(* Logix 5000 project; controller reports 1756-L63 rev 20.11; software revision 20.04; part 21 of 52 *)

        [1300].log_data[12].valid := 1, [1300].log_data[13].valid := 1, [1300].log_data[14].valid := 1, [1300].log_data[15].valid := 1, [1300].log_data[16].valid := 1, [1300].log_data[17].valid := 1, [1300].log_data[18].valid := 1, [1300].log_data[19].valid := 1, [1300].time.Year := 2023, [1300].time.Month := 1, [1300].time.Day := 14, [1300].time.Hour := 4, [1300].time.Minute := 44, [1300].time.Second := 59, [1301].log_data[0].min := 1.0, [1301].log_data[0].max := 1.0, [1301].log_data[0].total := 300.0, [1301].log_data[0].time := 300.0, [1301].log_data[0].minminute := 45, [1301].log_data[0].maxminute := 45, [1301].log_data[0].valid := 1, [1301].log_data[1].valid := 1, [1301].log_data[2].valid := 1, [1301].log_data[3].valid := 1, [1301].log_data[4].valid := 1, [1301].log_data[5].valid := 1, [1301].log_data[6].valid := 1, [1301].log_data[7].valid := 1, [1301].log_data[8].valid := 1, [1301].log_data[9].valid := 1, [1301].log_data[10].valid := 1, [1301].log_data[11].valid := 1, [1301].log_data[12].valid := 1, [1301].log_data[13].valid := 1, [1301].log_data[14].valid := 1, [1301].log_data[15].valid := 1, [1301].log_data[16].valid := 1, [1301].log_data[17].valid := 1, [1301].log_data[18].valid := 1, [1301].log_data[19].valid := 1, [1301].time.Year := 2023, [1301].time.Month := 1, [1301].time.Day := 14, [1301].time.Hour := 4, [1301].time.Minute := 49, [1301].time.Second := 59, [1302].log_data[0].min := 1.0, [1302].log_data[0].max := 1.0, [1302].log_data[0].total := 300.0, [1302].log_data[0].time := 300.0, [1302].log_data[0].minminute := 50, [1302].log_data[0].maxminute := 50, [1302].log_data[0].valid := 1, [1302].log_data[1].valid := 1, [1302].log_data[2].valid := 1, [1302].log_data[3].valid := 1, [1302].log_data[4].valid := 1, [1302].log_data[5].valid := 1, [1302].log_data[6].valid := 1, [1302].log_data[7].valid := 1,
        [1302].log_data[8].valid := 1, [1302].log_data[9].valid := 1, [1302].log_data[10].valid := 1, [1302].log_data[11].valid := 1, [1302].log_data[12].valid := 1, [1302].log_data[13].valid := 1, [1302].log_data[14].valid := 1, [1302].log_data[15].valid := 1, [1302].log_data[16].valid := 1, [1302].log_data[17].valid := 1, [1302].log_data[18].valid := 1, [1302].log_data[19].valid := 1, [1302].time.Year := 2023, [1302].time.Month := 1, [1302].time.Day := 14, [1302].time.Hour := 4, [1302].time.Minute := 54, [1302].time.Second := 59, [1303].log_data[0].min := 1.0, [1303].log_data[0].max := 1.0, [1303].log_data[0].total := 300.0, [1303].log_data[0].time := 300.0, [1303].log_data[0].minminute := 55, [1303].log_data[0].maxminute := 55, [1303].log_data[0].valid := 1, [1303].log_data[1].valid := 1, [1303].log_data[2].valid := 1, [1303].log_data[3].valid := 1, [1303].log_data[4].valid := 1, [1303].log_data[5].valid := 1, [1303].log_data[6].valid := 1, [1303].log_data[7].valid := 1, [1303].log_data[8].valid := 1, [1303].log_data[9].valid := 1, [1303].log_data[10].valid := 1, [1303].log_data[11].valid := 1, [1303].log_data[12].valid := 1, [1303].log_data[13].valid := 1, [1303].log_data[14].valid := 1, [1303].log_data[15].valid := 1, [1303].log_data[16].valid := 1, [1303].log_data[17].valid := 1, [1303].log_data[18].valid := 1, [1303].log_data[19].valid := 1, [1303].time.Year := 2023, [1303].time.Month := 1, [1303].time.Day := 14, [1303].time.Hour := 4, [1303].time.Minute := 59, [1303].time.Second := 59, [1304].log_data[0].min := 1.0, [1304].log_data[0].max := 1.0, [1304].log_data[0].total := 300.0, [1304].log_data[0].time := 300.0, [1304].log_data[0].valid := 1, [1304].log_data[1].valid := 1, [1304].log_data[2].valid := 1, [1304].log_data[3].valid := 1, [1304].log_data[4].valid := 1, [1304].log_data[5].valid := 1,
        [1304].log_data[6].valid := 1, [1304].log_data[7].valid := 1, [1304].log_data[8].valid := 1, [1304].log_data[9].valid := 1, [1304].log_data[10].valid := 1, [1304].log_data[11].valid := 1, [1304].log_data[12].valid := 1, [1304].log_data[13].valid := 1, [1304].log_data[14].valid := 1, [1304].log_data[15].valid := 1, [1304].log_data[16].valid := 1, [1304].log_data[17].valid := 1, [1304].log_data[18].valid := 1, [1304].log_data[19].valid := 1, [1304].time.Year := 2023, [1304].time.Month := 1, [1304].time.Day := 14, [1304].time.Hour := 5, [1304].time.Minute := 4, [1304].time.Second := 59, [1305].log_data[0].min := 1.0, [1305].log_data[0].max := 1.0, [1305].log_data[0].total := 300.0, [1305].log_data[0].time := 300.0, [1305].log_data[0].minminute := 5, [1305].log_data[0].maxminute := 5, [1305].log_data[0].valid := 1, [1305].log_data[1].valid := 1, [1305].log_data[2].valid := 1, [1305].log_data[3].valid := 1, [1305].log_data[4].valid := 1, [1305].log_data[5].valid := 1, [1305].log_data[6].valid := 1, [1305].log_data[7].valid := 1, [1305].log_data[8].valid := 1, [1305].log_data[9].valid := 1, [1305].log_data[10].valid := 1, [1305].log_data[11].valid := 1, [1305].log_data[12].valid := 1, [1305].log_data[13].valid := 1, [1305].log_data[14].valid := 1, [1305].log_data[15].valid := 1, [1305].log_data[16].valid := 1, [1305].log_data[17].valid := 1, [1305].log_data[18].valid := 1, [1305].log_data[19].valid := 1, [1305].time.Year := 2023, [1305].time.Month := 1, [1305].time.Day := 14, [1305].time.Hour := 5, [1305].time.Minute := 9, [1305].time.Second := 59, [1306].log_data[0].min := 1.0, [1306].log_data[0].max := 1.0, [1306].log_data[0].total := 300.0, [1306].log_data[0].time := 300.0, [1306].log_data[0].minminute := 10, [1306].log_data[0].maxminute := 10, [1306].log_data[0].valid := 1, [1306].log_data[1].valid := 1,
        [1306].log_data[2].valid := 1, [1306].log_data[3].valid := 1, [1306].log_data[4].valid := 1, [1306].log_data[5].valid := 1, [1306].log_data[6].valid := 1, [1306].log_data[7].valid := 1, [1306].log_data[8].valid := 1, [1306].log_data[9].valid := 1, [1306].log_data[10].valid := 1, [1306].log_data[11].valid := 1, [1306].log_data[12].valid := 1, [1306].log_data[13].valid := 1, [1306].log_data[14].valid := 1, [1306].log_data[15].valid := 1, [1306].log_data[16].valid := 1, [1306].log_data[17].valid := 1, [1306].log_data[18].valid := 1, [1306].log_data[19].valid := 1, [1306].time.Year := 2023, [1306].time.Month := 1, [1306].time.Day := 14, [1306].time.Hour := 5, [1306].time.Minute := 14, [1306].time.Second := 59, [1307].log_data[0].min := 1.0, [1307].log_data[0].max := 1.0, [1307].log_data[0].total := 300.0, [1307].log_data[0].time := 300.0, [1307].log_data[0].minminute := 15, [1307].log_data[0].maxminute := 15, [1307].log_data[0].valid := 1, [1307].log_data[1].valid := 1, [1307].log_data[2].valid := 1, [1307].log_data[3].valid := 1, [1307].log_data[4].valid := 1, [1307].log_data[5].valid := 1, [1307].log_data[6].valid := 1, [1307].log_data[7].valid := 1, [1307].log_data[8].valid := 1, [1307].log_data[9].valid := 1, [1307].log_data[10].valid := 1, [1307].log_data[11].valid := 1, [1307].log_data[12].valid := 1, [1307].log_data[13].valid := 1, [1307].log_data[14].valid := 1, [1307].log_data[15].valid := 1, [1307].log_data[16].valid := 1, [1307].log_data[17].valid := 1, [1307].log_data[18].valid := 1, [1307].log_data[19].valid := 1, [1307].time.Year := 2023, [1307].time.Month := 1, [1307].time.Day := 14, [1307].time.Hour := 5, [1307].time.Minute := 19, [1307].time.Second := 59, [1308].log_data[0].min := 1.0, [1308].log_data[0].max := 1.0, [1308].log_data[0].total := 300.0, [1308].log_data[0].time := 300.0,
        [1308].log_data[0].minminute := 20, [1308].log_data[0].maxminute := 20, [1308].log_data[0].valid := 1, [1308].log_data[1].valid := 1, [1308].log_data[2].valid := 1, [1308].log_data[3].valid := 1, [1308].log_data[4].valid := 1, [1308].log_data[5].valid := 1, [1308].log_data[6].valid := 1, [1308].log_data[7].valid := 1, [1308].log_data[8].valid := 1, [1308].log_data[9].valid := 1, [1308].log_data[10].valid := 1, [1308].log_data[11].valid := 1, [1308].log_data[12].valid := 1, [1308].log_data[13].valid := 1, [1308].log_data[14].valid := 1, [1308].log_data[15].valid := 1, [1308].log_data[16].valid := 1, [1308].log_data[17].valid := 1, [1308].log_data[18].valid := 1, [1308].log_data[19].valid := 1, [1308].time.Year := 2023, [1308].time.Month := 1, [1308].time.Day := 14, [1308].time.Hour := 5, [1308].time.Minute := 24, [1308].time.Second := 59, [1309].log_data[0].min := 1.0, [1309].log_data[0].max := 1.0, [1309].log_data[0].total := 300.0, [1309].log_data[0].time := 300.0, [1309].log_data[0].minminute := 25, [1309].log_data[0].maxminute := 25, [1309].log_data[0].valid := 1, [1309].log_data[1].valid := 1, [1309].log_data[2].valid := 1, [1309].log_data[3].valid := 1, [1309].log_data[4].valid := 1, [1309].log_data[5].valid := 1, [1309].log_data[6].valid := 1, [1309].log_data[7].valid := 1, [1309].log_data[8].valid := 1, [1309].log_data[9].valid := 1, [1309].log_data[10].valid := 1, [1309].log_data[11].valid := 1, [1309].log_data[12].valid := 1, [1309].log_data[13].valid := 1, [1309].log_data[14].valid := 1, [1309].log_data[15].valid := 1, [1309].log_data[16].valid := 1, [1309].log_data[17].valid := 1, [1309].log_data[18].valid := 1, [1309].log_data[19].valid := 1, [1309].time.Year := 2023, [1309].time.Month := 1, [1309].time.Day := 14, [1309].time.Hour := 5, [1309].time.Minute := 29, [1309].time.Second := 59,
        [1310].log_data[0].min := 1.0, [1310].log_data[0].max := 1.0, [1310].log_data[0].total := 300.0, [1310].log_data[0].time := 300.0, [1310].log_data[0].minminute := 30, [1310].log_data[0].maxminute := 30, [1310].log_data[0].valid := 1, [1310].log_data[1].valid := 1, [1310].log_data[2].valid := 1, [1310].log_data[3].valid := 1, [1310].log_data[4].valid := 1, [1310].log_data[5].valid := 1, [1310].log_data[6].valid := 1, [1310].log_data[7].valid := 1, [1310].log_data[8].valid := 1, [1310].log_data[9].valid := 1, [1310].log_data[10].valid := 1, [1310].log_data[11].valid := 1, [1310].log_data[12].valid := 1, [1310].log_data[13].valid := 1, [1310].log_data[14].valid := 1, [1310].log_data[15].valid := 1, [1310].log_data[16].valid := 1, [1310].log_data[17].valid := 1, [1310].log_data[18].valid := 1, [1310].log_data[19].valid := 1, [1310].time.Year := 2023, [1310].time.Month := 1, [1310].time.Day := 14, [1310].time.Hour := 5, [1310].time.Minute := 34, [1310].time.Second := 59, [1311].log_data[0].min := 1.0, [1311].log_data[0].max := 1.0, [1311].log_data[0].total := 300.0, [1311].log_data[0].time := 300.0, [1311].log_data[0].minminute := 35, [1311].log_data[0].maxminute := 35, [1311].log_data[0].valid := 1, [1311].log_data[1].valid := 1, [1311].log_data[2].valid := 1, [1311].log_data[3].valid := 1, [1311].log_data[4].valid := 1, [1311].log_data[5].valid := 1, [1311].log_data[6].valid := 1, [1311].log_data[7].valid := 1, [1311].log_data[8].valid := 1, [1311].log_data[9].valid := 1, [1311].log_data[10].valid := 1, [1311].log_data[11].valid := 1, [1311].log_data[12].valid := 1, [1311].log_data[13].valid := 1, [1311].log_data[14].valid := 1, [1311].log_data[15].valid := 1, [1311].log_data[16].valid := 1, [1311].log_data[17].valid := 1, [1311].log_data[18].valid := 1, [1311].log_data[19].valid := 1, [1311].time.Year := 2023, [1311].time.Month := 1,
        [1311].time.Day := 14, [1311].time.Hour := 5, [1311].time.Minute := 39, [1311].time.Second := 59, [1312].log_data[0].min := 1.0, [1312].log_data[0].max := 1.0, [1312].log_data[0].total := 300.0, [1312].log_data[0].time := 300.0, [1312].log_data[0].minminute := 40, [1312].log_data[0].maxminute := 40, [1312].log_data[0].valid := 1, [1312].log_data[1].valid := 1, [1312].log_data[2].valid := 1, [1312].log_data[3].valid := 1, [1312].log_data[4].valid := 1, [1312].log_data[5].valid := 1, [1312].log_data[6].valid := 1, [1312].log_data[7].valid := 1, [1312].log_data[8].valid := 1, [1312].log_data[9].valid := 1, [1312].log_data[10].valid := 1, [1312].log_data[11].valid := 1, [1312].log_data[12].valid := 1, [1312].log_data[13].valid := 1, [1312].log_data[14].valid := 1, [1312].log_data[15].valid := 1, [1312].log_data[16].valid := 1, [1312].log_data[17].valid := 1, [1312].log_data[18].valid := 1, [1312].log_data[19].valid := 1, [1312].time.Year := 2023, [1312].time.Month := 1, [1312].time.Day := 14, [1312].time.Hour := 5, [1312].time.Minute := 44, [1312].time.Second := 59, [1313].log_data[0].min := 1.0, [1313].log_data[0].max := 1.0, [1313].log_data[0].total := 300.0, [1313].log_data[0].time := 300.0, [1313].log_data[0].minminute := 45, [1313].log_data[0].maxminute := 45, [1313].log_data[0].valid := 1, [1313].log_data[1].valid := 1, [1313].log_data[2].valid := 1, [1313].log_data[3].valid := 1, [1313].log_data[4].valid := 1, [1313].log_data[5].valid := 1, [1313].log_data[6].valid := 1, [1313].log_data[7].valid := 1, [1313].log_data[8].valid := 1, [1313].log_data[9].valid := 1, [1313].log_data[10].valid := 1, [1313].log_data[11].valid := 1, [1313].log_data[12].valid := 1, [1313].log_data[13].valid := 1, [1313].log_data[14].valid := 1, [1313].log_data[15].valid := 1, [1313].log_data[16].valid := 1, [1313].log_data[17].valid := 1,
        [1313].log_data[18].valid := 1, [1313].log_data[19].valid := 1, [1313].time.Year := 2023, [1313].time.Month := 1, [1313].time.Day := 14, [1313].time.Hour := 5, [1313].time.Minute := 49, [1313].time.Second := 59, [1314].log_data[0].min := 1.0, [1314].log_data[0].max := 1.0, [1314].log_data[0].total := 300.0, [1314].log_data[0].time := 300.0, [1314].log_data[0].minminute := 50, [1314].log_data[0].maxminute := 50, [1314].log_data[0].valid := 1, [1314].log_data[1].valid := 1, [1314].log_data[2].valid := 1, [1314].log_data[3].valid := 1, [1314].log_data[4].valid := 1, [1314].log_data[5].valid := 1, [1314].log_data[6].valid := 1, [1314].log_data[7].valid := 1, [1314].log_data[8].valid := 1, [1314].log_data[9].valid := 1, [1314].log_data[10].valid := 1, [1314].log_data[11].valid := 1, [1314].log_data[12].valid := 1, [1314].log_data[13].valid := 1, [1314].log_data[14].valid := 1, [1314].log_data[15].valid := 1, [1314].log_data[16].valid := 1, [1314].log_data[17].valid := 1, [1314].log_data[18].valid := 1, [1314].log_data[19].valid := 1, [1314].time.Year := 2023, [1314].time.Month := 1, [1314].time.Day := 14, [1314].time.Hour := 5, [1314].time.Minute := 54, [1314].time.Second := 59, [1315].log_data[0].min := 1.0, [1315].log_data[0].max := 1.0, [1315].log_data[0].total := 300.0, [1315].log_data[0].time := 300.0, [1315].log_data[0].minminute := 55, [1315].log_data[0].maxminute := 55, [1315].log_data[0].valid := 1, [1315].log_data[1].valid := 1, [1315].log_data[2].valid := 1, [1315].log_data[3].valid := 1, [1315].log_data[4].valid := 1, [1315].log_data[5].valid := 1, [1315].log_data[6].valid := 1, [1315].log_data[7].valid := 1, [1315].log_data[8].valid := 1, [1315].log_data[9].valid := 1, [1315].log_data[10].valid := 1, [1315].log_data[11].valid := 1, [1315].log_data[12].valid := 1, [1315].log_data[13].valid := 1,
        [1315].log_data[14].valid := 1, [1315].log_data[15].valid := 1, [1315].log_data[16].valid := 1, [1315].log_data[17].valid := 1, [1315].log_data[18].valid := 1, [1315].log_data[19].valid := 1, [1315].time.Year := 2023, [1315].time.Month := 1, [1315].time.Day := 14, [1315].time.Hour := 5, [1315].time.Minute := 59, [1315].time.Second := 59, [1316].log_data[0].min := 1.0, [1316].log_data[0].max := 1.0, [1316].log_data[0].total := 300.0, [1316].log_data[0].time := 300.0, [1316].log_data[0].valid := 1, [1316].log_data[1].valid := 1, [1316].log_data[2].valid := 1, [1316].log_data[3].valid := 1, [1316].log_data[4].valid := 1, [1316].log_data[5].valid := 1, [1316].log_data[6].valid := 1, [1316].log_data[7].valid := 1, [1316].log_data[8].valid := 1, [1316].log_data[9].valid := 1, [1316].log_data[10].valid := 1, [1316].log_data[11].valid := 1, [1316].log_data[12].valid := 1, [1316].log_data[13].valid := 1, [1316].log_data[14].valid := 1, [1316].log_data[15].valid := 1, [1316].log_data[16].valid := 1, [1316].log_data[17].valid := 1, [1316].log_data[18].valid := 1, [1316].log_data[19].valid := 1, [1316].time.Year := 2023, [1316].time.Month := 1, [1316].time.Day := 14, [1316].time.Hour := 6, [1316].time.Minute := 4, [1316].time.Second := 59, [1317].log_data[0].min := 1.0, [1317].log_data[0].max := 1.0, [1317].log_data[0].total := 300.0, [1317].log_data[0].time := 300.0, [1317].log_data[0].minminute := 5, [1317].log_data[0].maxminute := 5, [1317].log_data[0].valid := 1, [1317].log_data[1].valid := 1, [1317].log_data[2].valid := 1, [1317].log_data[3].valid := 1, [1317].log_data[4].valid := 1, [1317].log_data[5].valid := 1, [1317].log_data[6].valid := 1, [1317].log_data[7].valid := 1, [1317].log_data[8].valid := 1, [1317].log_data[9].valid := 1, [1317].log_data[10].valid := 1, [1317].log_data[11].valid := 1,
        [1317].log_data[12].valid := 1, [1317].log_data[13].valid := 1, [1317].log_data[14].valid := 1, [1317].log_data[15].valid := 1, [1317].log_data[16].valid := 1, [1317].log_data[17].valid := 1, [1317].log_data[18].valid := 1, [1317].log_data[19].valid := 1, [1317].time.Year := 2023, [1317].time.Month := 1, [1317].time.Day := 14, [1317].time.Hour := 6, [1317].time.Minute := 9, [1317].time.Second := 59, [1318].log_data[0].min := 1.0, [1318].log_data[0].max := 1.0, [1318].log_data[0].total := 300.0, [1318].log_data[0].time := 300.0, [1318].log_data[0].minminute := 10, [1318].log_data[0].maxminute := 10, [1318].log_data[0].valid := 1, [1318].log_data[1].valid := 1, [1318].log_data[2].valid := 1, [1318].log_data[3].valid := 1, [1318].log_data[4].valid := 1, [1318].log_data[5].valid := 1, [1318].log_data[6].valid := 1, [1318].log_data[7].valid := 1, [1318].log_data[8].valid := 1, [1318].log_data[9].valid := 1, [1318].log_data[10].valid := 1, [1318].log_data[11].valid := 1, [1318].log_data[12].valid := 1, [1318].log_data[13].valid := 1, [1318].log_data[14].valid := 1, [1318].log_data[15].valid := 1, [1318].log_data[16].valid := 1, [1318].log_data[17].valid := 1, [1318].log_data[18].valid := 1, [1318].log_data[19].valid := 1, [1318].time.Year := 2023, [1318].time.Month := 1, [1318].time.Day := 14, [1318].time.Hour := 6, [1318].time.Minute := 14, [1318].time.Second := 59, [1319].log_data[0].min := 1.0, [1319].log_data[0].max := 1.0, [1319].log_data[0].total := 300.0, [1319].log_data[0].time := 300.0, [1319].log_data[0].minminute := 15, [1319].log_data[0].maxminute := 15, [1319].log_data[0].valid := 1, [1319].log_data[1].valid := 1, [1319].log_data[2].valid := 1, [1319].log_data[3].valid := 1, [1319].log_data[4].valid := 1, [1319].log_data[5].valid := 1, [1319].log_data[6].valid := 1, [1319].log_data[7].valid := 1,
        [1319].log_data[8].valid := 1, [1319].log_data[9].valid := 1, [1319].log_data[10].valid := 1, [1319].log_data[11].valid := 1, [1319].log_data[12].valid := 1, [1319].log_data[13].valid := 1, [1319].log_data[14].valid := 1, [1319].log_data[15].valid := 1, [1319].log_data[16].valid := 1, [1319].log_data[17].valid := 1, [1319].log_data[18].valid := 1, [1319].log_data[19].valid := 1, [1319].time.Year := 2023, [1319].time.Month := 1, [1319].time.Day := 14, [1319].time.Hour := 6, [1319].time.Minute := 19, [1319].time.Second := 59, [1320].log_data[0].min := 1.0, [1320].log_data[0].max := 1.0, [1320].log_data[0].total := 300.0, [1320].log_data[0].time := 300.0, [1320].log_data[0].minminute := 20, [1320].log_data[0].maxminute := 20, [1320].log_data[0].valid := 1, [1320].log_data[1].valid := 1, [1320].log_data[2].valid := 1, [1320].log_data[3].valid := 1, [1320].log_data[4].valid := 1, [1320].log_data[5].valid := 1, [1320].log_data[6].valid := 1, [1320].log_data[7].valid := 1, [1320].log_data[8].valid := 1, [1320].log_data[9].valid := 1, [1320].log_data[10].valid := 1, [1320].log_data[11].valid := 1, [1320].log_data[12].valid := 1, [1320].log_data[13].valid := 1, [1320].log_data[14].valid := 1, [1320].log_data[15].valid := 1, [1320].log_data[16].valid := 1, [1320].log_data[17].valid := 1, [1320].log_data[18].valid := 1, [1320].log_data[19].valid := 1, [1320].time.Year := 2023, [1320].time.Month := 1, [1320].time.Day := 14, [1320].time.Hour := 6, [1320].time.Minute := 24, [1320].time.Second := 59, [1321].log_data[0].min := 1.0, [1321].log_data[0].max := 1.0, [1321].log_data[0].total := 300.0, [1321].log_data[0].time := 300.0, [1321].log_data[0].minminute := 25, [1321].log_data[0].maxminute := 25, [1321].log_data[0].valid := 1, [1321].log_data[1].valid := 1, [1321].log_data[2].valid := 1, [1321].log_data[3].valid := 1,
        [1321].log_data[4].valid := 1, [1321].log_data[5].valid := 1, [1321].log_data[6].valid := 1, [1321].log_data[7].valid := 1, [1321].log_data[8].valid := 1, [1321].log_data[9].valid := 1, [1321].log_data[10].valid := 1, [1321].log_data[11].valid := 1, [1321].log_data[12].valid := 1, [1321].log_data[13].valid := 1, [1321].log_data[14].valid := 1, [1321].log_data[15].valid := 1, [1321].log_data[16].valid := 1, [1321].log_data[17].valid := 1, [1321].log_data[18].valid := 1, [1321].log_data[19].valid := 1, [1321].time.Year := 2023, [1321].time.Month := 1, [1321].time.Day := 14, [1321].time.Hour := 6, [1321].time.Minute := 29, [1321].time.Second := 59, [1322].log_data[0].min := 1.0, [1322].log_data[0].max := 1.0, [1322].log_data[0].total := 300.0, [1322].log_data[0].time := 300.0, [1322].log_data[0].minminute := 30, [1322].log_data[0].maxminute := 30, [1322].log_data[0].valid := 1, [1322].log_data[1].valid := 1, [1322].log_data[2].valid := 1, [1322].log_data[3].valid := 1, [1322].log_data[4].valid := 1, [1322].log_data[5].valid := 1, [1322].log_data[6].valid := 1, [1322].log_data[7].valid := 1, [1322].log_data[8].valid := 1, [1322].log_data[9].valid := 1, [1322].log_data[10].valid := 1, [1322].log_data[11].valid := 1, [1322].log_data[12].valid := 1, [1322].log_data[13].valid := 1, [1322].log_data[14].valid := 1, [1322].log_data[15].valid := 1, [1322].log_data[16].valid := 1, [1322].log_data[17].valid := 1, [1322].log_data[18].valid := 1, [1322].log_data[19].valid := 1, [1322].time.Year := 2023, [1322].time.Month := 1, [1322].time.Day := 14, [1322].time.Hour := 6, [1322].time.Minute := 34, [1322].time.Second := 59, [1323].log_data[0].min := 1.0, [1323].log_data[0].max := 1.0, [1323].log_data[0].total := 300.0, [1323].log_data[0].time := 300.0, [1323].log_data[0].minminute := 35, [1323].log_data[0].maxminute := 35,
        [1323].log_data[0].valid := 1, [1323].log_data[1].valid := 1, [1323].log_data[2].valid := 1, [1323].log_data[3].valid := 1, [1323].log_data[4].valid := 1, [1323].log_data[5].valid := 1, [1323].log_data[6].valid := 1, [1323].log_data[7].valid := 1, [1323].log_data[8].valid := 1, [1323].log_data[9].valid := 1, [1323].log_data[10].valid := 1, [1323].log_data[11].valid := 1, [1323].log_data[12].valid := 1, [1323].log_data[13].valid := 1, [1323].log_data[14].valid := 1, [1323].log_data[15].valid := 1, [1323].log_data[16].valid := 1, [1323].log_data[17].valid := 1, [1323].log_data[18].valid := 1, [1323].log_data[19].valid := 1, [1323].time.Year := 2023, [1323].time.Month := 1, [1323].time.Day := 14, [1323].time.Hour := 6, [1323].time.Minute := 39, [1323].time.Second := 59, [1324].log_data[0].min := 1.0, [1324].log_data[0].max := 1.0, [1324].log_data[0].total := 300.0, [1324].log_data[0].time := 300.0, [1324].log_data[0].minminute := 40, [1324].log_data[0].maxminute := 40, [1324].log_data[0].valid := 1, [1324].log_data[1].valid := 1, [1324].log_data[2].valid := 1, [1324].log_data[3].valid := 1, [1324].log_data[4].valid := 1, [1324].log_data[5].valid := 1, [1324].log_data[6].valid := 1, [1324].log_data[7].valid := 1, [1324].log_data[8].valid := 1, [1324].log_data[9].valid := 1, [1324].log_data[10].valid := 1, [1324].log_data[11].valid := 1, [1324].log_data[12].valid := 1, [1324].log_data[13].valid := 1, [1324].log_data[14].valid := 1, [1324].log_data[15].valid := 1, [1324].log_data[16].valid := 1, [1324].log_data[17].valid := 1, [1324].log_data[18].valid := 1, [1324].log_data[19].valid := 1, [1324].time.Year := 2023, [1324].time.Month := 1, [1324].time.Day := 14, [1324].time.Hour := 6, [1324].time.Minute := 44, [1324].time.Second := 59, [1325].log_data[0].min := 1.0, [1325].log_data[0].max := 1.0,
        [1325].log_data[0].total := 300.0, [1325].log_data[0].time := 300.0, [1325].log_data[0].minminute := 45, [1325].log_data[0].maxminute := 45, [1325].log_data[0].valid := 1, [1325].log_data[1].valid := 1, [1325].log_data[2].valid := 1, [1325].log_data[3].valid := 1, [1325].log_data[4].valid := 1, [1325].log_data[5].valid := 1, [1325].log_data[6].valid := 1, [1325].log_data[7].valid := 1, [1325].log_data[8].valid := 1, [1325].log_data[9].valid := 1, [1325].log_data[10].valid := 1, [1325].log_data[11].valid := 1, [1325].log_data[12].valid := 1, [1325].log_data[13].valid := 1, [1325].log_data[14].valid := 1, [1325].log_data[15].valid := 1, [1325].log_data[16].valid := 1, [1325].log_data[17].valid := 1, [1325].log_data[18].valid := 1, [1325].log_data[19].valid := 1, [1325].time.Year := 2023, [1325].time.Month := 1, [1325].time.Day := 14, [1325].time.Hour := 6, [1325].time.Minute := 49, [1325].time.Second := 59, [1326].log_data[0].min := 1.0, [1326].log_data[0].max := 1.0, [1326].log_data[0].total := 300.0, [1326].log_data[0].time := 300.0, [1326].log_data[0].minminute := 50, [1326].log_data[0].maxminute := 50, [1326].log_data[0].valid := 1, [1326].log_data[1].valid := 1, [1326].log_data[2].valid := 1, [1326].log_data[3].valid := 1, [1326].log_data[4].valid := 1, [1326].log_data[5].valid := 1, [1326].log_data[6].valid := 1, [1326].log_data[7].valid := 1, [1326].log_data[8].valid := 1, [1326].log_data[9].valid := 1, [1326].log_data[10].valid := 1, [1326].log_data[11].valid := 1, [1326].log_data[12].valid := 1, [1326].log_data[13].valid := 1, [1326].log_data[14].valid := 1, [1326].log_data[15].valid := 1, [1326].log_data[16].valid := 1, [1326].log_data[17].valid := 1, [1326].log_data[18].valid := 1, [1326].log_data[19].valid := 1, [1326].time.Year := 2023, [1326].time.Month := 1, [1326].time.Day := 14, [1326].time.Hour := 6,
        [1326].time.Minute := 54, [1326].time.Second := 59, [1327].log_data[0].min := 1.0, [1327].log_data[0].max := 1.0, [1327].log_data[0].total := 300.0, [1327].log_data[0].time := 300.0, [1327].log_data[0].minminute := 55, [1327].log_data[0].maxminute := 55, [1327].log_data[0].valid := 1, [1327].log_data[1].valid := 1, [1327].log_data[2].valid := 1, [1327].log_data[3].valid := 1, [1327].log_data[4].valid := 1, [1327].log_data[5].valid := 1, [1327].log_data[6].valid := 1, [1327].log_data[7].valid := 1, [1327].log_data[8].valid := 1, [1327].log_data[9].valid := 1, [1327].log_data[10].valid := 1, [1327].log_data[11].valid := 1, [1327].log_data[12].valid := 1, [1327].log_data[13].valid := 1, [1327].log_data[14].valid := 1, [1327].log_data[15].valid := 1, [1327].log_data[16].valid := 1, [1327].log_data[17].valid := 1, [1327].log_data[18].valid := 1, [1327].log_data[19].valid := 1, [1327].time.Year := 2023, [1327].time.Month := 1, [1327].time.Day := 14, [1327].time.Hour := 6, [1327].time.Minute := 59, [1327].time.Second := 59, [1328].log_data[0].min := 1.0, [1328].log_data[0].max := 1.0, [1328].log_data[0].total := 300.0, [1328].log_data[0].time := 300.0, [1328].log_data[0].valid := 1, [1328].log_data[1].valid := 1, [1328].log_data[2].valid := 1, [1328].log_data[3].valid := 1, [1328].log_data[4].valid := 1, [1328].log_data[5].valid := 1, [1328].log_data[6].valid := 1, [1328].log_data[7].valid := 1, [1328].log_data[8].valid := 1, [1328].log_data[9].valid := 1, [1328].log_data[10].valid := 1, [1328].log_data[11].valid := 1, [1328].log_data[12].valid := 1, [1328].log_data[13].valid := 1, [1328].log_data[14].valid := 1, [1328].log_data[15].valid := 1, [1328].log_data[16].valid := 1, [1328].log_data[17].valid := 1, [1328].log_data[18].valid := 1, [1328].log_data[19].valid := 1, [1328].time.Year := 2023, [1328].time.Month := 1,
        [1328].time.Day := 14, [1328].time.Hour := 7, [1328].time.Minute := 4, [1328].time.Second := 59, [1329].log_data[0].min := 1.0, [1329].log_data[0].max := 1.0, [1329].log_data[0].total := 300.0, [1329].log_data[0].time := 300.0, [1329].log_data[0].minminute := 5, [1329].log_data[0].maxminute := 5, [1329].log_data[0].valid := 1, [1329].log_data[1].valid := 1, [1329].log_data[2].valid := 1, [1329].log_data[3].valid := 1, [1329].log_data[4].valid := 1, [1329].log_data[5].valid := 1, [1329].log_data[6].valid := 1, [1329].log_data[7].valid := 1, [1329].log_data[8].valid := 1, [1329].log_data[9].valid := 1, [1329].log_data[10].valid := 1, [1329].log_data[11].valid := 1, [1329].log_data[12].valid := 1, [1329].log_data[13].valid := 1, [1329].log_data[14].valid := 1, [1329].log_data[15].valid := 1, [1329].log_data[16].valid := 1, [1329].log_data[17].valid := 1, [1329].log_data[18].valid := 1, [1329].log_data[19].valid := 1, [1329].time.Year := 2023, [1329].time.Month := 1, [1329].time.Day := 14, [1329].time.Hour := 7, [1329].time.Minute := 9, [1329].time.Second := 59, [1330].log_data[0].min := 1.0, [1330].log_data[0].max := 1.0, [1330].log_data[0].total := 300.0, [1330].log_data[0].time := 300.0, [1330].log_data[0].minminute := 10, [1330].log_data[0].maxminute := 10, [1330].log_data[0].valid := 1, [1330].log_data[1].valid := 1, [1330].log_data[2].valid := 1, [1330].log_data[3].valid := 1, [1330].log_data[4].valid := 1, [1330].log_data[5].valid := 1, [1330].log_data[6].valid := 1, [1330].log_data[7].valid := 1, [1330].log_data[8].valid := 1, [1330].log_data[9].valid := 1, [1330].log_data[10].valid := 1, [1330].log_data[11].valid := 1, [1330].log_data[12].valid := 1, [1330].log_data[13].valid := 1, [1330].log_data[14].valid := 1, [1330].log_data[15].valid := 1, [1330].log_data[16].valid := 1, [1330].log_data[17].valid := 1,
        [1330].log_data[18].valid := 1, [1330].log_data[19].valid := 1, [1330].time.Year := 2023, [1330].time.Month := 1, [1330].time.Day := 14, [1330].time.Hour := 7, [1330].time.Minute := 14, [1330].time.Second := 59, [1331].log_data[0].min := 1.0, [1331].log_data[0].max := 1.0, [1331].log_data[0].total := 300.0, [1331].log_data[0].time := 300.0, [1331].log_data[0].minminute := 15, [1331].log_data[0].maxminute := 15, [1331].log_data[0].valid := 1, [1331].log_data[1].valid := 1, [1331].log_data[2].valid := 1, [1331].log_data[3].valid := 1, [1331].log_data[4].valid := 1, [1331].log_data[5].valid := 1, [1331].log_data[6].valid := 1, [1331].log_data[7].valid := 1, [1331].log_data[8].valid := 1, [1331].log_data[9].valid := 1, [1331].log_data[10].valid := 1, [1331].log_data[11].valid := 1, [1331].log_data[12].valid := 1, [1331].log_data[13].valid := 1, [1331].log_data[14].valid := 1, [1331].log_data[15].valid := 1, [1331].log_data[16].valid := 1, [1331].log_data[17].valid := 1, [1331].log_data[18].valid := 1, [1331].log_data[19].valid := 1, [1331].time.Year := 2023, [1331].time.Month := 1, [1331].time.Day := 14, [1331].time.Hour := 7, [1331].time.Minute := 19, [1331].time.Second := 59, [1332].log_data[0].min := 1.0, [1332].log_data[0].max := 1.0, [1332].log_data[0].total := 300.0, [1332].log_data[0].time := 300.0, [1332].log_data[0].minminute := 20, [1332].log_data[0].maxminute := 20, [1332].log_data[0].valid := 1, [1332].log_data[1].valid := 1, [1332].log_data[2].valid := 1, [1332].log_data[3].valid := 1, [1332].log_data[4].valid := 1, [1332].log_data[5].valid := 1, [1332].log_data[6].valid := 1, [1332].log_data[7].valid := 1, [1332].log_data[8].valid := 1, [1332].log_data[9].valid := 1, [1332].log_data[10].valid := 1, [1332].log_data[11].valid := 1, [1332].log_data[12].valid := 1, [1332].log_data[13].valid := 1,
        [1332].log_data[14].valid := 1, [1332].log_data[15].valid := 1, [1332].log_data[16].valid := 1, [1332].log_data[17].valid := 1, [1332].log_data[18].valid := 1, [1332].log_data[19].valid := 1, [1332].time.Year := 2023, [1332].time.Month := 1, [1332].time.Day := 14, [1332].time.Hour := 7, [1332].time.Minute := 24, [1332].time.Second := 59, [1333].log_data[0].min := 1.0, [1333].log_data[0].max := 1.0, [1333].log_data[0].total := 300.0, [1333].log_data[0].time := 300.0, [1333].log_data[0].minminute := 25, [1333].log_data[0].maxminute := 25, [1333].log_data[0].valid := 1, [1333].log_data[1].valid := 1, [1333].log_data[2].valid := 1, [1333].log_data[3].valid := 1, [1333].log_data[4].valid := 1, [1333].log_data[5].valid := 1, [1333].log_data[6].valid := 1, [1333].log_data[7].valid := 1, [1333].log_data[8].valid := 1, [1333].log_data[9].valid := 1, [1333].log_data[10].valid := 1, [1333].log_data[11].valid := 1, [1333].log_data[12].valid := 1, [1333].log_data[13].valid := 1, [1333].log_data[14].valid := 1, [1333].log_data[15].valid := 1, [1333].log_data[16].valid := 1, [1333].log_data[17].valid := 1, [1333].log_data[18].valid := 1, [1333].log_data[19].valid := 1, [1333].time.Year := 2023, [1333].time.Month := 1, [1333].time.Day := 14, [1333].time.Hour := 7, [1333].time.Minute := 29, [1333].time.Second := 59, [1334].log_data[0].min := 1.0, [1334].log_data[0].max := 1.0, [1334].log_data[0].total := 300.0, [1334].log_data[0].time := 300.0, [1334].log_data[0].minminute := 30, [1334].log_data[0].maxminute := 30, [1334].log_data[0].valid := 1, [1334].log_data[1].valid := 1, [1334].log_data[2].valid := 1, [1334].log_data[3].valid := 1, [1334].log_data[4].valid := 1, [1334].log_data[5].valid := 1, [1334].log_data[6].valid := 1, [1334].log_data[7].valid := 1, [1334].log_data[8].valid := 1, [1334].log_data[9].valid := 1,
        [1334].log_data[10].valid := 1, [1334].log_data[11].valid := 1, [1334].log_data[12].valid := 1, [1334].log_data[13].valid := 1, [1334].log_data[14].valid := 1, [1334].log_data[15].valid := 1, [1334].log_data[16].valid := 1, [1334].log_data[17].valid := 1, [1334].log_data[18].valid := 1, [1334].log_data[19].valid := 1, [1334].time.Year := 2023, [1334].time.Month := 1, [1334].time.Day := 14, [1334].time.Hour := 7, [1334].time.Minute := 34, [1334].time.Second := 59, [1335].log_data[0].min := 1.0, [1335].log_data[0].max := 1.0, [1335].log_data[0].total := 300.0, [1335].log_data[0].time := 300.0, [1335].log_data[0].minminute := 35, [1335].log_data[0].maxminute := 35, [1335].log_data[0].valid := 1, [1335].log_data[1].valid := 1, [1335].log_data[2].valid := 1, [1335].log_data[3].valid := 1, [1335].log_data[4].valid := 1, [1335].log_data[5].valid := 1, [1335].log_data[6].valid := 1, [1335].log_data[7].valid := 1, [1335].log_data[8].valid := 1, [1335].log_data[9].valid := 1, [1335].log_data[10].valid := 1, [1335].log_data[11].valid := 1, [1335].log_data[12].valid := 1, [1335].log_data[13].valid := 1, [1335].log_data[14].valid := 1, [1335].log_data[15].valid := 1, [1335].log_data[16].valid := 1, [1335].log_data[17].valid := 1, [1335].log_data[18].valid := 1, [1335].log_data[19].valid := 1, [1335].time.Year := 2023, [1335].time.Month := 1, [1335].time.Day := 14, [1335].time.Hour := 7, [1335].time.Minute := 39, [1335].time.Second := 59, [1336].log_data[0].min := 1.0, [1336].log_data[0].max := 1.0, [1336].log_data[0].total := 300.0, [1336].log_data[0].time := 300.0, [1336].log_data[0].minminute := 40, [1336].log_data[0].maxminute := 40, [1336].log_data[0].valid := 1, [1336].log_data[1].valid := 1, [1336].log_data[2].valid := 1, [1336].log_data[3].valid := 1, [1336].log_data[4].valid := 1, [1336].log_data[5].valid := 1,
        [1336].log_data[6].valid := 1, [1336].log_data[7].valid := 1, [1336].log_data[8].valid := 1, [1336].log_data[9].valid := 1, [1336].log_data[10].valid := 1, [1336].log_data[11].valid := 1, [1336].log_data[12].valid := 1, [1336].log_data[13].valid := 1, [1336].log_data[14].valid := 1, [1336].log_data[15].valid := 1, [1336].log_data[16].valid := 1, [1336].log_data[17].valid := 1, [1336].log_data[18].valid := 1, [1336].log_data[19].valid := 1, [1336].time.Year := 2023, [1336].time.Month := 1, [1336].time.Day := 14, [1336].time.Hour := 7, [1336].time.Minute := 44, [1336].time.Second := 59, [1337].log_data[0].min := 1.0, [1337].log_data[0].max := 1.0, [1337].log_data[0].total := 300.0, [1337].log_data[0].time := 300.0, [1337].log_data[0].minminute := 45, [1337].log_data[0].maxminute := 45, [1337].log_data[0].valid := 1, [1337].log_data[1].valid := 1, [1337].log_data[2].valid := 1, [1337].log_data[3].valid := 1, [1337].log_data[4].valid := 1, [1337].log_data[5].valid := 1, [1337].log_data[6].valid := 1, [1337].log_data[7].valid := 1, [1337].log_data[8].valid := 1, [1337].log_data[9].valid := 1, [1337].log_data[10].valid := 1, [1337].log_data[11].valid := 1, [1337].log_data[12].valid := 1, [1337].log_data[13].valid := 1, [1337].log_data[14].valid := 1, [1337].log_data[15].valid := 1, [1337].log_data[16].valid := 1, [1337].log_data[17].valid := 1, [1337].log_data[18].valid := 1, [1337].log_data[19].valid := 1, [1337].time.Year := 2023, [1337].time.Month := 1, [1337].time.Day := 14, [1337].time.Hour := 7, [1337].time.Minute := 49, [1337].time.Second := 59, [1338].log_data[0].min := 1.0, [1338].log_data[0].max := 1.0, [1338].log_data[0].total := 300.0, [1338].log_data[0].time := 300.0, [1338].log_data[0].minminute := 50, [1338].log_data[0].maxminute := 50, [1338].log_data[0].valid := 1, [1338].log_data[1].valid := 1,
        [1338].log_data[2].valid := 1, [1338].log_data[3].valid := 1, [1338].log_data[4].valid := 1, [1338].log_data[5].valid := 1, [1338].log_data[6].valid := 1, [1338].log_data[7].valid := 1, [1338].log_data[8].valid := 1, [1338].log_data[9].valid := 1, [1338].log_data[10].valid := 1, [1338].log_data[11].valid := 1, [1338].log_data[12].valid := 1, [1338].log_data[13].valid := 1, [1338].log_data[14].valid := 1, [1338].log_data[15].valid := 1, [1338].log_data[16].valid := 1, [1338].log_data[17].valid := 1, [1338].log_data[18].valid := 1, [1338].log_data[19].valid := 1, [1338].time.Year := 2023, [1338].time.Month := 1, [1338].time.Day := 14, [1338].time.Hour := 7, [1338].time.Minute := 54, [1338].time.Second := 59, [1339].log_data[0].min := 1.0, [1339].log_data[0].max := 1.0, [1339].log_data[0].total := 300.0, [1339].log_data[0].time := 300.0, [1339].log_data[0].minminute := 55, [1339].log_data[0].maxminute := 55, [1339].log_data[0].valid := 1, [1339].log_data[1].valid := 1, [1339].log_data[2].valid := 1, [1339].log_data[3].valid := 1, [1339].log_data[4].valid := 1, [1339].log_data[5].valid := 1, [1339].log_data[6].valid := 1, [1339].log_data[7].valid := 1, [1339].log_data[8].valid := 1, [1339].log_data[9].valid := 1, [1339].log_data[10].valid := 1, [1339].log_data[11].valid := 1, [1339].log_data[12].valid := 1, [1339].log_data[13].valid := 1, [1339].log_data[14].valid := 1, [1339].log_data[15].valid := 1, [1339].log_data[16].valid := 1, [1339].log_data[17].valid := 1, [1339].log_data[18].valid := 1, [1339].log_data[19].valid := 1, [1339].time.Year := 2023, [1339].time.Month := 1, [1339].time.Day := 14, [1339].time.Hour := 7, [1339].time.Minute := 59, [1339].time.Second := 59, [1340].log_data[0].min := 1.0, [1340].log_data[0].max := 1.0, [1340].log_data[0].total := 300.0, [1340].log_data[0].time := 300.0,
        [1340].log_data[0].valid := 1, [1340].log_data[1].valid := 1, [1340].log_data[2].valid := 1, [1340].log_data[3].valid := 1, [1340].log_data[4].valid := 1, [1340].log_data[5].valid := 1, [1340].log_data[6].valid := 1, [1340].log_data[7].valid := 1, [1340].log_data[8].valid := 1, [1340].log_data[9].valid := 1, [1340].log_data[10].valid := 1, [1340].log_data[11].valid := 1, [1340].log_data[12].valid := 1, [1340].log_data[13].valid := 1, [1340].log_data[14].valid := 1, [1340].log_data[15].valid := 1, [1340].log_data[16].valid := 1, [1340].log_data[17].valid := 1, [1340].log_data[18].valid := 1, [1340].log_data[19].valid := 1, [1340].time.Year := 2023, [1340].time.Month := 1, [1340].time.Day := 14, [1340].time.Hour := 8, [1340].time.Minute := 4, [1340].time.Second := 59, [1341].log_data[0].min := 1.0, [1341].log_data[0].max := 1.0, [1341].log_data[0].total := 300.0, [1341].log_data[0].time := 300.0, [1341].log_data[0].minminute := 5, [1341].log_data[0].maxminute := 5, [1341].log_data[0].valid := 1, [1341].log_data[1].valid := 1, [1341].log_data[2].valid := 1, [1341].log_data[3].valid := 1, [1341].log_data[4].valid := 1, [1341].log_data[5].valid := 1, [1341].log_data[6].valid := 1, [1341].log_data[7].valid := 1, [1341].log_data[8].valid := 1, [1341].log_data[9].valid := 1, [1341].log_data[10].valid := 1, [1341].log_data[11].valid := 1, [1341].log_data[12].valid := 1, [1341].log_data[13].valid := 1, [1341].log_data[14].valid := 1, [1341].log_data[15].valid := 1, [1341].log_data[16].valid := 1, [1341].log_data[17].valid := 1, [1341].log_data[18].valid := 1, [1341].log_data[19].valid := 1, [1341].time.Year := 2023, [1341].time.Month := 1, [1341].time.Day := 14, [1341].time.Hour := 8, [1341].time.Minute := 9, [1341].time.Second := 59, [1342].log_data[0].min := 1.0, [1342].log_data[0].max := 1.0,
        [1342].log_data[0].total := 300.0, [1342].log_data[0].time := 300.0, [1342].log_data[0].minminute := 10, [1342].log_data[0].maxminute := 10, [1342].log_data[0].valid := 1, [1342].log_data[1].valid := 1, [1342].log_data[2].valid := 1, [1342].log_data[3].valid := 1, [1342].log_data[4].valid := 1, [1342].log_data[5].valid := 1, [1342].log_data[6].valid := 1, [1342].log_data[7].valid := 1, [1342].log_data[8].valid := 1, [1342].log_data[9].valid := 1, [1342].log_data[10].valid := 1, [1342].log_data[11].valid := 1, [1342].log_data[12].valid := 1, [1342].log_data[13].valid := 1, [1342].log_data[14].valid := 1, [1342].log_data[15].valid := 1, [1342].log_data[16].valid := 1, [1342].log_data[17].valid := 1, [1342].log_data[18].valid := 1, [1342].log_data[19].valid := 1, [1342].time.Year := 2023, [1342].time.Month := 1, [1342].time.Day := 14, [1342].time.Hour := 8, [1342].time.Minute := 14, [1342].time.Second := 59, [1343].log_data[0].min := 1.0, [1343].log_data[0].max := 1.0, [1343].log_data[0].total := 300.0, [1343].log_data[0].time := 300.0, [1343].log_data[0].minminute := 15, [1343].log_data[0].maxminute := 15, [1343].log_data[0].valid := 1, [1343].log_data[1].valid := 1, [1343].log_data[2].valid := 1, [1343].log_data[3].valid := 1, [1343].log_data[4].valid := 1, [1343].log_data[5].valid := 1, [1343].log_data[6].valid := 1, [1343].log_data[7].valid := 1, [1343].log_data[8].valid := 1, [1343].log_data[9].valid := 1, [1343].log_data[10].valid := 1, [1343].log_data[11].valid := 1, [1343].log_data[12].valid := 1, [1343].log_data[13].valid := 1, [1343].log_data[14].valid := 1, [1343].log_data[15].valid := 1, [1343].log_data[16].valid := 1, [1343].log_data[17].valid := 1, [1343].log_data[18].valid := 1, [1343].log_data[19].valid := 1, [1343].time.Year := 2023, [1343].time.Month := 1, [1343].time.Day := 14, [1343].time.Hour := 8,
        [1343].time.Minute := 19, [1343].time.Second := 59, [1344].log_data[0].min := 1.0, [1344].log_data[0].max := 1.0, [1344].log_data[0].total := 300.0, [1344].log_data[0].time := 300.0, [1344].log_data[0].minminute := 20, [1344].log_data[0].maxminute := 20, [1344].log_data[0].valid := 1, [1344].log_data[1].valid := 1, [1344].log_data[2].valid := 1, [1344].log_data[3].valid := 1, [1344].log_data[4].valid := 1, [1344].log_data[5].valid := 1, [1344].log_data[6].valid := 1, [1344].log_data[7].valid := 1, [1344].log_data[8].valid := 1, [1344].log_data[9].valid := 1, [1344].log_data[10].valid := 1, [1344].log_data[11].valid := 1, [1344].log_data[12].valid := 1, [1344].log_data[13].valid := 1, [1344].log_data[14].valid := 1, [1344].log_data[15].valid := 1, [1344].log_data[16].valid := 1, [1344].log_data[17].valid := 1, [1344].log_data[18].valid := 1, [1344].log_data[19].valid := 1, [1344].time.Year := 2023, [1344].time.Month := 1, [1344].time.Day := 14, [1344].time.Hour := 8, [1344].time.Minute := 24, [1344].time.Second := 59, [1345].log_data[0].min := 1.0, [1345].log_data[0].max := 1.0, [1345].log_data[0].total := 300.0, [1345].log_data[0].time := 300.0, [1345].log_data[0].minminute := 25, [1345].log_data[0].maxminute := 25, [1345].log_data[0].valid := 1, [1345].log_data[1].valid := 1, [1345].log_data[2].valid := 1, [1345].log_data[3].valid := 1, [1345].log_data[4].valid := 1, [1345].log_data[5].valid := 1, [1345].log_data[6].valid := 1, [1345].log_data[7].valid := 1, [1345].log_data[8].valid := 1, [1345].log_data[9].valid := 1, [1345].log_data[10].valid := 1, [1345].log_data[11].valid := 1, [1345].log_data[12].valid := 1, [1345].log_data[13].valid := 1, [1345].log_data[14].valid := 1, [1345].log_data[15].valid := 1, [1345].log_data[16].valid := 1, [1345].log_data[17].valid := 1, [1345].log_data[18].valid := 1, [1345].log_data[19].valid := 1,
        [1345].time.Year := 2023, [1345].time.Month := 1, [1345].time.Day := 14, [1345].time.Hour := 8, [1345].time.Minute := 29, [1345].time.Second := 59, [1346].log_data[0].min := 1.0, [1346].log_data[0].max := 1.0, [1346].log_data[0].total := 300.0, [1346].log_data[0].time := 300.0, [1346].log_data[0].minminute := 30, [1346].log_data[0].maxminute := 30, [1346].log_data[0].valid := 1, [1346].log_data[1].valid := 1, [1346].log_data[2].valid := 1, [1346].log_data[3].valid := 1, [1346].log_data[4].valid := 1, [1346].log_data[5].valid := 1, [1346].log_data[6].valid := 1, [1346].log_data[7].valid := 1, [1346].log_data[8].valid := 1, [1346].log_data[9].valid := 1, [1346].log_data[10].valid := 1, [1346].log_data[11].valid := 1, [1346].log_data[12].valid := 1, [1346].log_data[13].valid := 1, [1346].log_data[14].valid := 1, [1346].log_data[15].valid := 1, [1346].log_data[16].valid := 1, [1346].log_data[17].valid := 1, [1346].log_data[18].valid := 1, [1346].log_data[19].valid := 1, [1346].time.Year := 2023, [1346].time.Month := 1, [1346].time.Day := 14, [1346].time.Hour := 8, [1346].time.Minute := 34, [1346].time.Second := 59, [1347].log_data[0].min := 1.0, [1347].log_data[0].max := 1.0, [1347].log_data[0].total := 300.0, [1347].log_data[0].time := 300.0, [1347].log_data[0].minminute := 35, [1347].log_data[0].maxminute := 35, [1347].log_data[0].valid := 1, [1347].log_data[1].valid := 1, [1347].log_data[2].valid := 1, [1347].log_data[3].valid := 1, [1347].log_data[4].valid := 1, [1347].log_data[5].valid := 1, [1347].log_data[6].valid := 1, [1347].log_data[7].valid := 1, [1347].log_data[8].valid := 1, [1347].log_data[9].valid := 1, [1347].log_data[10].valid := 1, [1347].log_data[11].valid := 1, [1347].log_data[12].valid := 1, [1347].log_data[13].valid := 1, [1347].log_data[14].valid := 1, [1347].log_data[15].valid := 1,
        [1347].log_data[16].valid := 1, [1347].log_data[17].valid := 1, [1347].log_data[18].valid := 1, [1347].log_data[19].valid := 1, [1347].time.Year := 2023, [1347].time.Month := 1, [1347].time.Day := 14, [1347].time.Hour := 8, [1347].time.Minute := 39, [1347].time.Second := 59, [1348].log_data[0].min := 1.0, [1348].log_data[0].max := 1.0, [1348].log_data[0].total := 300.0, [1348].log_data[0].time := 300.0, [1348].log_data[0].minminute := 40, [1348].log_data[0].maxminute := 40, [1348].log_data[0].valid := 1, [1348].log_data[1].valid := 1, [1348].log_data[2].valid := 1, [1348].log_data[3].valid := 1, [1348].log_data[4].valid := 1, [1348].log_data[5].valid := 1, [1348].log_data[6].valid := 1, [1348].log_data[7].valid := 1, [1348].log_data[8].valid := 1, [1348].log_data[9].valid := 1, [1348].log_data[10].valid := 1, [1348].log_data[11].valid := 1, [1348].log_data[12].valid := 1, [1348].log_data[13].valid := 1, [1348].log_data[14].valid := 1, [1348].log_data[15].valid := 1, [1348].log_data[16].valid := 1, [1348].log_data[17].valid := 1, [1348].log_data[18].valid := 1, [1348].log_data[19].valid := 1, [1348].time.Year := 2023, [1348].time.Month := 1, [1348].time.Day := 14, [1348].time.Hour := 8, [1348].time.Minute := 44, [1348].time.Second := 59, [1349].log_data[0].min := 1.0, [1349].log_data[0].max := 1.0, [1349].log_data[0].total := 300.0, [1349].log_data[0].time := 300.0, [1349].log_data[0].minminute := 45, [1349].log_data[0].maxminute := 45, [1349].log_data[0].valid := 1, [1349].log_data[1].valid := 1, [1349].log_data[2].valid := 1, [1349].log_data[3].valid := 1, [1349].log_data[4].valid := 1, [1349].log_data[5].valid := 1, [1349].log_data[6].valid := 1, [1349].log_data[7].valid := 1, [1349].log_data[8].valid := 1, [1349].log_data[9].valid := 1, [1349].log_data[10].valid := 1, [1349].log_data[11].valid := 1,
        [1349].log_data[12].valid := 1, [1349].log_data[13].valid := 1, [1349].log_data[14].valid := 1, [1349].log_data[15].valid := 1, [1349].log_data[16].valid := 1, [1349].log_data[17].valid := 1, [1349].log_data[18].valid := 1, [1349].log_data[19].valid := 1, [1349].time.Year := 2023, [1349].time.Month := 1, [1349].time.Day := 14, [1349].time.Hour := 8, [1349].time.Minute := 49, [1349].time.Second := 59, [1350].log_data[0].min := 1.0, [1350].log_data[0].max := 1.0, [1350].log_data[0].total := 300.0, [1350].log_data[0].time := 300.0, [1350].log_data[0].minminute := 50, [1350].log_data[0].maxminute := 50, [1350].log_data[0].valid := 1, [1350].log_data[1].valid := 1, [1350].log_data[2].valid := 1, [1350].log_data[3].valid := 1, [1350].log_data[4].valid := 1, [1350].log_data[5].valid := 1, [1350].log_data[6].valid := 1, [1350].log_data[7].valid := 1, [1350].log_data[8].valid := 1, [1350].log_data[9].valid := 1, [1350].log_data[10].valid := 1, [1350].log_data[11].valid := 1, [1350].log_data[12].valid := 1, [1350].log_data[13].valid := 1, [1350].log_data[14].valid := 1, [1350].log_data[15].valid := 1, [1350].log_data[16].valid := 1, [1350].log_data[17].valid := 1, [1350].log_data[18].valid := 1, [1350].log_data[19].valid := 1, [1350].time.Year := 2023, [1350].time.Month := 1, [1350].time.Day := 14, [1350].time.Hour := 8, [1350].time.Minute := 54, [1350].time.Second := 59, [1351].log_data[0].min := 1.0, [1351].log_data[0].max := 1.0, [1351].log_data[0].total := 300.0, [1351].log_data[0].time := 300.0, [1351].log_data[0].minminute := 55, [1351].log_data[0].maxminute := 55, [1351].log_data[0].valid := 1, [1351].log_data[1].valid := 1, [1351].log_data[2].valid := 1, [1351].log_data[3].valid := 1, [1351].log_data[4].valid := 1, [1351].log_data[5].valid := 1, [1351].log_data[6].valid := 1, [1351].log_data[7].valid := 1,
        [1351].log_data[8].valid := 1, [1351].log_data[9].valid := 1, [1351].log_data[10].valid := 1, [1351].log_data[11].valid := 1, [1351].log_data[12].valid := 1, [1351].log_data[13].valid := 1, [1351].log_data[14].valid := 1, [1351].log_data[15].valid := 1, [1351].log_data[16].valid := 1, [1351].log_data[17].valid := 1, [1351].log_data[18].valid := 1, [1351].log_data[19].valid := 1, [1351].time.Year := 2023, [1351].time.Month := 1, [1351].time.Day := 14, [1351].time.Hour := 8, [1351].time.Minute := 59, [1351].time.Second := 59, [1352].log_data[0].min := 1.0, [1352].log_data[0].max := 1.0, [1352].log_data[0].total := 300.0, [1352].log_data[0].time := 300.0, [1352].log_data[0].valid := 1, [1352].log_data[1].valid := 1, [1352].log_data[2].valid := 1, [1352].log_data[3].valid := 1, [1352].log_data[4].valid := 1, [1352].log_data[5].valid := 1, [1352].log_data[6].valid := 1, [1352].log_data[7].valid := 1, [1352].log_data[8].valid := 1, [1352].log_data[9].valid := 1, [1352].log_data[10].valid := 1, [1352].log_data[11].valid := 1, [1352].log_data[12].valid := 1, [1352].log_data[13].valid := 1, [1352].log_data[14].valid := 1, [1352].log_data[15].valid := 1, [1352].log_data[16].valid := 1, [1352].log_data[17].valid := 1, [1352].log_data[18].valid := 1, [1352].log_data[19].valid := 1, [1352].time.Year := 2023, [1352].time.Month := 1, [1352].time.Day := 14, [1352].time.Hour := 9, [1352].time.Minute := 4, [1352].time.Second := 59, [1353].log_data[0].min := 1.0, [1353].log_data[0].max := 1.0, [1353].log_data[0].total := 300.0, [1353].log_data[0].time := 300.0, [1353].log_data[0].minminute := 5, [1353].log_data[0].maxminute := 5, [1353].log_data[0].valid := 1, [1353].log_data[1].valid := 1, [1353].log_data[2].valid := 1, [1353].log_data[3].valid := 1, [1353].log_data[4].valid := 1, [1353].log_data[5].valid := 1,
        [1353].log_data[6].valid := 1, [1353].log_data[7].valid := 1, [1353].log_data[8].valid := 1, [1353].log_data[9].valid := 1, [1353].log_data[10].valid := 1, [1353].log_data[11].valid := 1, [1353].log_data[12].valid := 1, [1353].log_data[13].valid := 1, [1353].log_data[14].valid := 1, [1353].log_data[15].valid := 1, [1353].log_data[16].valid := 1, [1353].log_data[17].valid := 1, [1353].log_data[18].valid := 1, [1353].log_data[19].valid := 1, [1353].time.Year := 2023, [1353].time.Month := 1, [1353].time.Day := 14, [1353].time.Hour := 9, [1353].time.Minute := 9, [1353].time.Second := 59, [1354].log_data[0].min := 1.0, [1354].log_data[0].max := 1.0, [1354].log_data[0].total := 300.0, [1354].log_data[0].time := 300.0, [1354].log_data[0].minminute := 10, [1354].log_data[0].maxminute := 10, [1354].log_data[0].valid := 1, [1354].log_data[1].valid := 1, [1354].log_data[2].valid := 1, [1354].log_data[3].valid := 1, [1354].log_data[4].valid := 1, [1354].log_data[5].valid := 1, [1354].log_data[6].valid := 1, [1354].log_data[7].valid := 1, [1354].log_data[8].valid := 1, [1354].log_data[9].valid := 1, [1354].log_data[10].valid := 1, [1354].log_data[11].valid := 1, [1354].log_data[12].valid := 1, [1354].log_data[13].valid := 1, [1354].log_data[14].valid := 1, [1354].log_data[15].valid := 1, [1354].log_data[16].valid := 1, [1354].log_data[17].valid := 1, [1354].log_data[18].valid := 1, [1354].log_data[19].valid := 1, [1354].time.Year := 2023, [1354].time.Month := 1, [1354].time.Day := 14, [1354].time.Hour := 9, [1354].time.Minute := 14, [1354].time.Second := 59, [1355].log_data[0].min := 1.0, [1355].log_data[0].max := 1.0, [1355].log_data[0].total := 300.0, [1355].log_data[0].time := 300.0, [1355].log_data[0].minminute := 15, [1355].log_data[0].maxminute := 15, [1355].log_data[0].valid := 1, [1355].log_data[1].valid := 1,
        [1355].log_data[2].valid := 1, [1355].log_data[3].valid := 1, [1355].log_data[4].valid := 1, [1355].log_data[5].valid := 1, [1355].log_data[6].valid := 1, [1355].log_data[7].valid := 1, [1355].log_data[8].valid := 1, [1355].log_data[9].valid := 1, [1355].log_data[10].valid := 1, [1355].log_data[11].valid := 1, [1355].log_data[12].valid := 1, [1355].log_data[13].valid := 1, [1355].log_data[14].valid := 1, [1355].log_data[15].valid := 1, [1355].log_data[16].valid := 1, [1355].log_data[17].valid := 1, [1355].log_data[18].valid := 1, [1355].log_data[19].valid := 1, [1355].time.Year := 2023, [1355].time.Month := 1, [1355].time.Day := 14, [1355].time.Hour := 9, [1355].time.Minute := 19, [1355].time.Second := 59, [1356].log_data[0].min := 1.0, [1356].log_data[0].max := 1.0, [1356].log_data[0].total := 300.0, [1356].log_data[0].time := 300.0, [1356].log_data[0].minminute := 20, [1356].log_data[0].maxminute := 20, [1356].log_data[0].valid := 1, [1356].log_data[1].valid := 1, [1356].log_data[2].valid := 1, [1356].log_data[3].valid := 1, [1356].log_data[4].valid := 1, [1356].log_data[5].valid := 1, [1356].log_data[6].valid := 1, [1356].log_data[7].valid := 1, [1356].log_data[8].valid := 1, [1356].log_data[9].valid := 1, [1356].log_data[10].valid := 1, [1356].log_data[11].valid := 1, [1356].log_data[12].valid := 1, [1356].log_data[13].valid := 1, [1356].log_data[14].valid := 1, [1356].log_data[15].valid := 1, [1356].log_data[16].valid := 1, [1356].log_data[17].valid := 1, [1356].log_data[18].valid := 1, [1356].log_data[19].valid := 1, [1356].time.Year := 2023, [1356].time.Month := 1, [1356].time.Day := 14, [1356].time.Hour := 9, [1356].time.Minute := 24, [1356].time.Second := 59, [1357].log_data[0].min := 1.0, [1357].log_data[0].max := 1.0, [1357].log_data[0].total := 300.0, [1357].log_data[0].time := 300.0,
        [1357].log_data[0].minminute := 25, [1357].log_data[0].maxminute := 25, [1357].log_data[0].valid := 1, [1357].log_data[1].valid := 1, [1357].log_data[2].valid := 1, [1357].log_data[3].valid := 1, [1357].log_data[4].valid := 1, [1357].log_data[5].valid := 1, [1357].log_data[6].valid := 1, [1357].log_data[7].valid := 1, [1357].log_data[8].valid := 1, [1357].log_data[9].valid := 1, [1357].log_data[10].valid := 1, [1357].log_data[11].valid := 1, [1357].log_data[12].valid := 1, [1357].log_data[13].valid := 1, [1357].log_data[14].valid := 1, [1357].log_data[15].valid := 1, [1357].log_data[16].valid := 1, [1357].log_data[17].valid := 1, [1357].log_data[18].valid := 1, [1357].log_data[19].valid := 1, [1357].time.Year := 2023, [1357].time.Month := 1, [1357].time.Day := 14, [1357].time.Hour := 9, [1357].time.Minute := 29, [1357].time.Second := 59, [1358].log_data[0].min := 1.0, [1358].log_data[0].max := 1.0, [1358].log_data[0].total := 300.0, [1358].log_data[0].time := 300.0, [1358].log_data[0].minminute := 30, [1358].log_data[0].maxminute := 30, [1358].log_data[0].valid := 1, [1358].log_data[1].valid := 1, [1358].log_data[2].valid := 1, [1358].log_data[3].valid := 1, [1358].log_data[4].valid := 1, [1358].log_data[5].valid := 1, [1358].log_data[6].valid := 1, [1358].log_data[7].valid := 1, [1358].log_data[8].valid := 1, [1358].log_data[9].valid := 1, [1358].log_data[10].valid := 1, [1358].log_data[11].valid := 1, [1358].log_data[12].valid := 1, [1358].log_data[13].valid := 1, [1358].log_data[14].valid := 1, [1358].log_data[15].valid := 1, [1358].log_data[16].valid := 1, [1358].log_data[17].valid := 1, [1358].log_data[18].valid := 1, [1358].log_data[19].valid := 1, [1358].time.Year := 2023, [1358].time.Month := 1, [1358].time.Day := 14, [1358].time.Hour := 9, [1358].time.Minute := 34, [1358].time.Second := 59,
        [1359].log_data[0].min := 1.0, [1359].log_data[0].max := 1.0, [1359].log_data[0].total := 300.0, [1359].log_data[0].time := 300.0, [1359].log_data[0].minminute := 35, [1359].log_data[0].maxminute := 35, [1359].log_data[0].valid := 1, [1359].log_data[1].valid := 1, [1359].log_data[2].valid := 1, [1359].log_data[3].valid := 1, [1359].log_data[4].valid := 1, [1359].log_data[5].valid := 1, [1359].log_data[6].valid := 1, [1359].log_data[7].valid := 1, [1359].log_data[8].valid := 1, [1359].log_data[9].valid := 1, [1359].log_data[10].valid := 1, [1359].log_data[11].valid := 1, [1359].log_data[12].valid := 1, [1359].log_data[13].valid := 1, [1359].log_data[14].valid := 1, [1359].log_data[15].valid := 1, [1359].log_data[16].valid := 1, [1359].log_data[17].valid := 1, [1359].log_data[18].valid := 1, [1359].log_data[19].valid := 1, [1359].time.Year := 2023, [1359].time.Month := 1, [1359].time.Day := 14, [1359].time.Hour := 9, [1359].time.Minute := 39, [1359].time.Second := 59, [1360].log_data[0].min := 1.0, [1360].log_data[0].max := 1.0, [1360].log_data[0].total := 300.0, [1360].log_data[0].time := 300.0, [1360].log_data[0].minminute := 40, [1360].log_data[0].maxminute := 40, [1360].log_data[0].valid := 1, [1360].log_data[1].valid := 1, [1360].log_data[2].valid := 1, [1360].log_data[3].valid := 1, [1360].log_data[4].valid := 1, [1360].log_data[5].valid := 1, [1360].log_data[6].valid := 1, [1360].log_data[7].valid := 1, [1360].log_data[8].valid := 1, [1360].log_data[9].valid := 1, [1360].log_data[10].valid := 1, [1360].log_data[11].valid := 1, [1360].log_data[12].valid := 1, [1360].log_data[13].valid := 1, [1360].log_data[14].valid := 1, [1360].log_data[15].valid := 1, [1360].log_data[16].valid := 1, [1360].log_data[17].valid := 1, [1360].log_data[18].valid := 1, [1360].log_data[19].valid := 1, [1360].time.Year := 2023, [1360].time.Month := 1,
        [1360].time.Day := 14, [1360].time.Hour := 9, [1360].time.Minute := 44, [1360].time.Second := 59, [1361].log_data[0].min := 1.0, [1361].log_data[0].max := 1.0, [1361].log_data[0].total := 300.0, [1361].log_data[0].time := 300.0, [1361].log_data[0].minminute := 45, [1361].log_data[0].maxminute := 45, [1361].log_data[0].valid := 1, [1361].log_data[1].valid := 1, [1361].log_data[2].valid := 1, [1361].log_data[3].valid := 1, [1361].log_data[4].valid := 1, [1361].log_data[5].valid := 1, [1361].log_data[6].valid := 1, [1361].log_data[7].valid := 1, [1361].log_data[8].valid := 1, [1361].log_data[9].valid := 1, [1361].log_data[10].valid := 1, [1361].log_data[11].valid := 1, [1361].log_data[12].valid := 1, [1361].log_data[13].valid := 1, [1361].log_data[14].valid := 1, [1361].log_data[15].valid := 1, [1361].log_data[16].valid := 1, [1361].log_data[17].valid := 1, [1361].log_data[18].valid := 1, [1361].log_data[19].valid := 1, [1361].time.Year := 2023, [1361].time.Month := 1, [1361].time.Day := 14, [1361].time.Hour := 9, [1361].time.Minute := 49, [1361].time.Second := 59, [1362].log_data[0].min := 1.0, [1362].log_data[0].max := 1.0, [1362].log_data[0].total := 300.0, [1362].log_data[0].time := 300.0, [1362].log_data[0].minminute := 50, [1362].log_data[0].maxminute := 50, [1362].log_data[0].valid := 1, [1362].log_data[1].valid := 1, [1362].log_data[2].valid := 1, [1362].log_data[3].valid := 1, [1362].log_data[4].valid := 1, [1362].log_data[5].valid := 1, [1362].log_data[6].valid := 1, [1362].log_data[7].valid := 1, [1362].log_data[8].valid := 1, [1362].log_data[9].valid := 1, [1362].log_data[10].valid := 1, [1362].log_data[11].valid := 1, [1362].log_data[12].valid := 1, [1362].log_data[13].valid := 1, [1362].log_data[14].valid := 1, [1362].log_data[15].valid := 1, [1362].log_data[16].valid := 1, [1362].log_data[17].valid := 1,
        [1362].log_data[18].valid := 1, [1362].log_data[19].valid := 1, [1362].time.Year := 2023, [1362].time.Month := 1, [1362].time.Day := 14, [1362].time.Hour := 9, [1362].time.Minute := 54, [1362].time.Second := 59, [1363].log_data[0].min := 1.0, [1363].log_data[0].max := 1.0, [1363].log_data[0].total := 300.0, [1363].log_data[0].time := 300.0, [1363].log_data[0].minminute := 55, [1363].log_data[0].maxminute := 55, [1363].log_data[0].valid := 1, [1363].log_data[1].valid := 1, [1363].log_data[2].valid := 1, [1363].log_data[3].valid := 1, [1363].log_data[4].valid := 1, [1363].log_data[5].valid := 1, [1363].log_data[6].valid := 1, [1363].log_data[7].valid := 1, [1363].log_data[8].valid := 1, [1363].log_data[9].valid := 1, [1363].log_data[10].valid := 1, [1363].log_data[11].valid := 1, [1363].log_data[12].valid := 1, [1363].log_data[13].valid := 1, [1363].log_data[14].valid := 1, [1363].log_data[15].valid := 1, [1363].log_data[16].valid := 1, [1363].log_data[17].valid := 1, [1363].log_data[18].valid := 1, [1363].log_data[19].valid := 1, [1363].time.Year := 2023, [1363].time.Month := 1, [1363].time.Day := 14, [1363].time.Hour := 9, [1363].time.Minute := 59, [1363].time.Second := 59, [1364].log_data[0].min := 1.0, [1364].log_data[0].max := 1.0, [1364].log_data[0].total := 300.0, [1364].log_data[0].time := 300.0, [1364].log_data[0].valid := 1, [1364].log_data[1].valid := 1, [1364].log_data[2].valid := 1, [1364].log_data[3].valid := 1, [1364].log_data[4].valid := 1, [1364].log_data[5].valid := 1, [1364].log_data[6].valid := 1, [1364].log_data[7].valid := 1, [1364].log_data[8].valid := 1, [1364].log_data[9].valid := 1, [1364].log_data[10].valid := 1, [1364].log_data[11].valid := 1, [1364].log_data[12].valid := 1, [1364].log_data[13].valid := 1, [1364].log_data[14].valid := 1, [1364].log_data[15].valid := 1,
        [1364].log_data[16].valid := 1, [1364].log_data[17].valid := 1, [1364].log_data[18].valid := 1, [1364].log_data[19].valid := 1, [1364].time.Year := 2023, [1364].time.Month := 1, [1364].time.Day := 14, [1364].time.Hour := 10, [1364].time.Minute := 4, [1364].time.Second := 59, [1365].log_data[0].min := 1.0, [1365].log_data[0].max := 1.0, [1365].log_data[0].total := 300.0, [1365].log_data[0].time := 300.0, [1365].log_data[0].minminute := 5, [1365].log_data[0].maxminute := 5, [1365].log_data[0].valid := 1, [1365].log_data[1].valid := 1, [1365].log_data[2].valid := 1, [1365].log_data[3].valid := 1, [1365].log_data[4].valid := 1, [1365].log_data[5].valid := 1, [1365].log_data[6].valid := 1, [1365].log_data[7].valid := 1, [1365].log_data[8].valid := 1, [1365].log_data[9].valid := 1, [1365].log_data[10].valid := 1, [1365].log_data[11].valid := 1, [1365].log_data[12].valid := 1, [1365].log_data[13].valid := 1, [1365].log_data[14].valid := 1, [1365].log_data[15].valid := 1, [1365].log_data[16].valid := 1, [1365].log_data[17].valid := 1, [1365].log_data[18].valid := 1, [1365].log_data[19].valid := 1, [1365].time.Year := 2023, [1365].time.Month := 1, [1365].time.Day := 14, [1365].time.Hour := 10, [1365].time.Minute := 9, [1365].time.Second := 59, [1366].log_data[0].min := 1.0, [1366].log_data[0].max := 1.0, [1366].log_data[0].total := 300.0, [1366].log_data[0].time := 300.0, [1366].log_data[0].minminute := 10, [1366].log_data[0].maxminute := 10, [1366].log_data[0].valid := 1, [1366].log_data[1].valid := 1, [1366].log_data[2].valid := 1, [1366].log_data[3].valid := 1, [1366].log_data[4].valid := 1, [1366].log_data[5].valid := 1, [1366].log_data[6].valid := 1, [1366].log_data[7].valid := 1, [1366].log_data[8].valid := 1, [1366].log_data[9].valid := 1, [1366].log_data[10].valid := 1, [1366].log_data[11].valid := 1,
        [1366].log_data[12].valid := 1, [1366].log_data[13].valid := 1, [1366].log_data[14].valid := 1, [1366].log_data[15].valid := 1, [1366].log_data[16].valid := 1, [1366].log_data[17].valid := 1, [1366].log_data[18].valid := 1, [1366].log_data[19].valid := 1, [1366].time.Year := 2023, [1366].time.Month := 1, [1366].time.Day := 14, [1366].time.Hour := 10, [1366].time.Minute := 14, [1366].time.Second := 59, [1367].log_data[0].min := 1.0, [1367].log_data[0].max := 1.0, [1367].log_data[0].total := 300.0, [1367].log_data[0].time := 300.0, [1367].log_data[0].minminute := 15, [1367].log_data[0].maxminute := 15, [1367].log_data[0].valid := 1, [1367].log_data[1].valid := 1, [1367].log_data[2].valid := 1, [1367].log_data[3].valid := 1, [1367].log_data[4].valid := 1, [1367].log_data[5].valid := 1, [1367].log_data[6].valid := 1, [1367].log_data[7].valid := 1, [1367].log_data[8].valid := 1, [1367].log_data[9].valid := 1, [1367].log_data[10].valid := 1, [1367].log_data[11].valid := 1, [1367].log_data[12].valid := 1, [1367].log_data[13].valid := 1, [1367].log_data[14].valid := 1, [1367].log_data[15].valid := 1, [1367].log_data[16].valid := 1, [1367].log_data[17].valid := 1, [1367].log_data[18].valid := 1, [1367].log_data[19].valid := 1, [1367].time.Year := 2023, [1367].time.Month := 1, [1367].time.Day := 14, [1367].time.Hour := 10, [1367].time.Minute := 19, [1367].time.Second := 59, [1368].log_data[0].min := 1.0, [1368].log_data[0].max := 1.0, [1368].log_data[0].total := 300.0, [1368].log_data[0].time := 300.0, [1368].log_data[0].minminute := 20, [1368].log_data[0].maxminute := 20, [1368].log_data[0].valid := 1, [1368].log_data[1].valid := 1, [1368].log_data[2].valid := 1, [1368].log_data[3].valid := 1, [1368].log_data[4].valid := 1, [1368].log_data[5].valid := 1, [1368].log_data[6].valid := 1, [1368].log_data[7].valid := 1,
        [1368].log_data[8].valid := 1, [1368].log_data[9].valid := 1, [1368].log_data[10].valid := 1, [1368].log_data[11].valid := 1, [1368].log_data[12].valid := 1, [1368].log_data[13].valid := 1, [1368].log_data[14].valid := 1, [1368].log_data[15].valid := 1, [1368].log_data[16].valid := 1, [1368].log_data[17].valid := 1, [1368].log_data[18].valid := 1, [1368].log_data[19].valid := 1, [1368].time.Year := 2023, [1368].time.Month := 1, [1368].time.Day := 14, [1368].time.Hour := 10, [1368].time.Minute := 24, [1368].time.Second := 59, [1369].log_data[0].min := 1.0, [1369].log_data[0].max := 1.0, [1369].log_data[0].total := 300.0, [1369].log_data[0].time := 300.0, [1369].log_data[0].minminute := 25, [1369].log_data[0].maxminute := 25, [1369].log_data[0].valid := 1, [1369].log_data[1].valid := 1, [1369].log_data[2].valid := 1, [1369].log_data[3].valid := 1, [1369].log_data[4].valid := 1, [1369].log_data[5].valid := 1, [1369].log_data[6].valid := 1, [1369].log_data[7].valid := 1, [1369].log_data[8].valid := 1, [1369].log_data[9].valid := 1, [1369].log_data[10].valid := 1, [1369].log_data[11].valid := 1, [1369].log_data[12].valid := 1, [1369].log_data[13].valid := 1, [1369].log_data[14].valid := 1, [1369].log_data[15].valid := 1, [1369].log_data[16].valid := 1, [1369].log_data[17].valid := 1, [1369].log_data[18].valid := 1, [1369].log_data[19].valid := 1, [1369].time.Year := 2023, [1369].time.Month := 1, [1369].time.Day := 14, [1369].time.Hour := 10, [1369].time.Minute := 29, [1369].time.Second := 59, [1370].log_data[0].min := 1.0, [1370].log_data[0].max := 1.0, [1370].log_data[0].total := 300.0, [1370].log_data[0].time := 300.0, [1370].log_data[0].minminute := 30, [1370].log_data[0].maxminute := 30, [1370].log_data[0].valid := 1, [1370].log_data[1].valid := 1, [1370].log_data[2].valid := 1, [1370].log_data[3].valid := 1,
        [1370].log_data[4].valid := 1, [1370].log_data[5].valid := 1, [1370].log_data[6].valid := 1, [1370].log_data[7].valid := 1, [1370].log_data[8].valid := 1, [1370].log_data[9].valid := 1, [1370].log_data[10].valid := 1, [1370].log_data[11].valid := 1, [1370].log_data[12].valid := 1, [1370].log_data[13].valid := 1, [1370].log_data[14].valid := 1, [1370].log_data[15].valid := 1, [1370].log_data[16].valid := 1, [1370].log_data[17].valid := 1, [1370].log_data[18].valid := 1, [1370].log_data[19].valid := 1, [1370].time.Year := 2023, [1370].time.Month := 1, [1370].time.Day := 14, [1370].time.Hour := 10, [1370].time.Minute := 34, [1370].time.Second := 59, [1371].log_data[0].min := 1.0, [1371].log_data[0].max := 1.0, [1371].log_data[0].total := 300.0, [1371].log_data[0].time := 300.0, [1371].log_data[0].minminute := 35, [1371].log_data[0].maxminute := 35, [1371].log_data[0].valid := 1, [1371].log_data[1].valid := 1, [1371].log_data[2].valid := 1, [1371].log_data[3].valid := 1, [1371].log_data[4].valid := 1, [1371].log_data[5].valid := 1, [1371].log_data[6].valid := 1, [1371].log_data[7].valid := 1, [1371].log_data[8].valid := 1, [1371].log_data[9].valid := 1, [1371].log_data[10].valid := 1, [1371].log_data[11].valid := 1, [1371].log_data[12].valid := 1, [1371].log_data[13].valid := 1, [1371].log_data[14].valid := 1, [1371].log_data[15].valid := 1, [1371].log_data[16].valid := 1, [1371].log_data[17].valid := 1, [1371].log_data[18].valid := 1, [1371].log_data[19].valid := 1, [1371].time.Year := 2023, [1371].time.Month := 1, [1371].time.Day := 14, [1371].time.Hour := 10, [1371].time.Minute := 39, [1371].time.Second := 59, [1372].log_data[0].min := 1.0, [1372].log_data[0].max := 1.0, [1372].log_data[0].total := 300.0, [1372].log_data[0].time := 300.0, [1372].log_data[0].minminute := 40, [1372].log_data[0].maxminute := 40,
        [1372].log_data[0].valid := 1, [1372].log_data[1].valid := 1, [1372].log_data[2].valid := 1, [1372].log_data[3].valid := 1, [1372].log_data[4].valid := 1, [1372].log_data[5].valid := 1, [1372].log_data[6].valid := 1, [1372].log_data[7].valid := 1, [1372].log_data[8].valid := 1, [1372].log_data[9].valid := 1, [1372].log_data[10].valid := 1, [1372].log_data[11].valid := 1, [1372].log_data[12].valid := 1, [1372].log_data[13].valid := 1, [1372].log_data[14].valid := 1, [1372].log_data[15].valid := 1, [1372].log_data[16].valid := 1, [1372].log_data[17].valid := 1, [1372].log_data[18].valid := 1, [1372].log_data[19].valid := 1, [1372].time.Year := 2023, [1372].time.Month := 1, [1372].time.Day := 14, [1372].time.Hour := 10, [1372].time.Minute := 44, [1372].time.Second := 59, [1373].log_data[0].min := 1.0, [1373].log_data[0].max := 1.0, [1373].log_data[0].total := 300.0, [1373].log_data[0].time := 300.0, [1373].log_data[0].minminute := 45, [1373].log_data[0].maxminute := 45, [1373].log_data[0].valid := 1, [1373].log_data[1].valid := 1, [1373].log_data[2].valid := 1, [1373].log_data[3].valid := 1, [1373].log_data[4].valid := 1, [1373].log_data[5].valid := 1, [1373].log_data[6].valid := 1, [1373].log_data[7].valid := 1, [1373].log_data[8].valid := 1, [1373].log_data[9].valid := 1, [1373].log_data[10].valid := 1, [1373].log_data[11].valid := 1, [1373].log_data[12].valid := 1, [1373].log_data[13].valid := 1, [1373].log_data[14].valid := 1, [1373].log_data[15].valid := 1, [1373].log_data[16].valid := 1, [1373].log_data[17].valid := 1, [1373].log_data[18].valid := 1, [1373].log_data[19].valid := 1, [1373].time.Year := 2023, [1373].time.Month := 1, [1373].time.Day := 14, [1373].time.Hour := 10, [1373].time.Minute := 49, [1373].time.Second := 59, [1374].log_data[0].min := 1.0, [1374].log_data[0].max := 1.0,
        [1374].log_data[0].total := 300.0, [1374].log_data[0].time := 300.0, [1374].log_data[0].minminute := 50, [1374].log_data[0].maxminute := 50, [1374].log_data[0].valid := 1, [1374].log_data[1].valid := 1, [1374].log_data[2].valid := 1, [1374].log_data[3].valid := 1, [1374].log_data[4].valid := 1, [1374].log_data[5].valid := 1, [1374].log_data[6].valid := 1, [1374].log_data[7].valid := 1, [1374].log_data[8].valid := 1, [1374].log_data[9].valid := 1, [1374].log_data[10].valid := 1, [1374].log_data[11].valid := 1, [1374].log_data[12].valid := 1, [1374].log_data[13].valid := 1, [1374].log_data[14].valid := 1, [1374].log_data[15].valid := 1, [1374].log_data[16].valid := 1, [1374].log_data[17].valid := 1, [1374].log_data[18].valid := 1, [1374].log_data[19].valid := 1, [1374].time.Year := 2023, [1374].time.Month := 1, [1374].time.Day := 14, [1374].time.Hour := 10, [1374].time.Minute := 54, [1374].time.Second := 59, [1375].log_data[0].min := 1.0, [1375].log_data[0].max := 1.0, [1375].log_data[0].total := 300.0, [1375].log_data[0].time := 300.0, [1375].log_data[0].minminute := 55, [1375].log_data[0].maxminute := 55, [1375].log_data[0].valid := 1, [1375].log_data[1].valid := 1, [1375].log_data[2].valid := 1, [1375].log_data[3].valid := 1, [1375].log_data[4].valid := 1, [1375].log_data[5].valid := 1, [1375].log_data[6].valid := 1, [1375].log_data[7].valid := 1, [1375].log_data[8].valid := 1, [1375].log_data[9].valid := 1, [1375].log_data[10].valid := 1, [1375].log_data[11].valid := 1, [1375].log_data[12].valid := 1, [1375].log_data[13].valid := 1, [1375].log_data[14].valid := 1, [1375].log_data[15].valid := 1, [1375].log_data[16].valid := 1, [1375].log_data[17].valid := 1, [1375].log_data[18].valid := 1, [1375].log_data[19].valid := 1, [1375].time.Year := 2023, [1375].time.Month := 1, [1375].time.Day := 14, [1375].time.Hour := 10,
        [1375].time.Minute := 59, [1375].time.Second := 59, [1376].log_data[0].min := 1.0, [1376].log_data[0].max := 1.0, [1376].log_data[0].total := 300.0, [1376].log_data[0].time := 300.0, [1376].log_data[0].valid := 1, [1376].log_data[1].valid := 1, [1376].log_data[2].valid := 1, [1376].log_data[3].valid := 1, [1376].log_data[4].valid := 1, [1376].log_data[5].valid := 1, [1376].log_data[6].valid := 1, [1376].log_data[7].valid := 1, [1376].log_data[8].valid := 1, [1376].log_data[9].valid := 1, [1376].log_data[10].valid := 1, [1376].log_data[11].valid := 1, [1376].log_data[12].valid := 1, [1376].log_data[13].valid := 1, [1376].log_data[14].valid := 1, [1376].log_data[15].valid := 1, [1376].log_data[16].valid := 1, [1376].log_data[17].valid := 1, [1376].log_data[18].valid := 1, [1376].log_data[19].valid := 1, [1376].time.Year := 2023, [1376].time.Month := 1, [1376].time.Day := 14, [1376].time.Hour := 11, [1376].time.Minute := 4, [1376].time.Second := 59, [1377].log_data[0].min := 1.0, [1377].log_data[0].max := 1.0, [1377].log_data[0].total := 300.0, [1377].log_data[0].time := 300.0, [1377].log_data[0].minminute := 5, [1377].log_data[0].maxminute := 5, [1377].log_data[0].valid := 1, [1377].log_data[1].valid := 1, [1377].log_data[2].valid := 1, [1377].log_data[3].valid := 1, [1377].log_data[4].valid := 1, [1377].log_data[5].valid := 1, [1377].log_data[6].valid := 1, [1377].log_data[7].valid := 1, [1377].log_data[8].valid := 1, [1377].log_data[9].valid := 1, [1377].log_data[10].valid := 1, [1377].log_data[11].valid := 1, [1377].log_data[12].valid := 1, [1377].log_data[13].valid := 1, [1377].log_data[14].valid := 1, [1377].log_data[15].valid := 1, [1377].log_data[16].valid := 1, [1377].log_data[17].valid := 1, [1377].log_data[18].valid := 1, [1377].log_data[19].valid := 1, [1377].time.Year := 2023, [1377].time.Month := 1,
        [1377].time.Day := 14, [1377].time.Hour := 11, [1377].time.Minute := 9, [1377].time.Second := 59, [1378].log_data[0].min := 1.0, [1378].log_data[0].max := 1.0, [1378].log_data[0].total := 300.0, [1378].log_data[0].time := 300.0, [1378].log_data[0].minminute := 10, [1378].log_data[0].maxminute := 10, [1378].log_data[0].valid := 1, [1378].log_data[1].valid := 1, [1378].log_data[2].valid := 1, [1378].log_data[3].valid := 1, [1378].log_data[4].valid := 1, [1378].log_data[5].valid := 1, [1378].log_data[6].valid := 1, [1378].log_data[7].valid := 1, [1378].log_data[8].valid := 1, [1378].log_data[9].valid := 1, [1378].log_data[10].valid := 1, [1378].log_data[11].valid := 1, [1378].log_data[12].valid := 1, [1378].log_data[13].valid := 1, [1378].log_data[14].valid := 1, [1378].log_data[15].valid := 1, [1378].log_data[16].valid := 1, [1378].log_data[17].valid := 1, [1378].log_data[18].valid := 1, [1378].log_data[19].valid := 1, [1378].time.Year := 2023, [1378].time.Month := 1, [1378].time.Day := 14, [1378].time.Hour := 11, [1378].time.Minute := 14, [1378].time.Second := 59, [1379].log_data[0].min := 1.0, [1379].log_data[0].max := 1.0, [1379].log_data[0].total := 300.0, [1379].log_data[0].time := 300.0, [1379].log_data[0].minminute := 15, [1379].log_data[0].maxminute := 15, [1379].log_data[0].valid := 1, [1379].log_data[1].valid := 1, [1379].log_data[2].valid := 1, [1379].log_data[3].valid := 1, [1379].log_data[4].valid := 1, [1379].log_data[5].valid := 1, [1379].log_data[6].valid := 1, [1379].log_data[7].valid := 1, [1379].log_data[8].valid := 1, [1379].log_data[9].valid := 1, [1379].log_data[10].valid := 1, [1379].log_data[11].valid := 1, [1379].log_data[12].valid := 1, [1379].log_data[13].valid := 1, [1379].log_data[14].valid := 1, [1379].log_data[15].valid := 1, [1379].log_data[16].valid := 1, [1379].log_data[17].valid := 1,
        [1379].log_data[18].valid := 1, [1379].log_data[19].valid := 1, [1379].time.Year := 2023, [1379].time.Month := 1, [1379].time.Day := 14, [1379].time.Hour := 11, [1379].time.Minute := 19, [1379].time.Second := 59, [1380].log_data[0].min := 1.0, [1380].log_data[0].max := 1.0, [1380].log_data[0].total := 300.0, [1380].log_data[0].time := 300.0, [1380].log_data[0].minminute := 20, [1380].log_data[0].maxminute := 20, [1380].log_data[0].valid := 1, [1380].log_data[1].valid := 1, [1380].log_data[2].valid := 1, [1380].log_data[3].valid := 1, [1380].log_data[4].valid := 1, [1380].log_data[5].valid := 1, [1380].log_data[6].valid := 1, [1380].log_data[7].valid := 1, [1380].log_data[8].valid := 1, [1380].log_data[9].valid := 1, [1380].log_data[10].valid := 1, [1380].log_data[11].valid := 1, [1380].log_data[12].valid := 1, [1380].log_data[13].valid := 1, [1380].log_data[14].valid := 1, [1380].log_data[15].valid := 1, [1380].log_data[16].valid := 1, [1380].log_data[17].valid := 1, [1380].log_data[18].valid := 1, [1380].log_data[19].valid := 1, [1380].time.Year := 2023, [1380].time.Month := 1, [1380].time.Day := 14, [1380].time.Hour := 11, [1380].time.Minute := 24, [1380].time.Second := 59, [1381].log_data[0].min := 1.0, [1381].log_data[0].max := 1.0, [1381].log_data[0].total := 300.0, [1381].log_data[0].time := 300.0, [1381].log_data[0].minminute := 25, [1381].log_data[0].maxminute := 25, [1381].log_data[0].valid := 1, [1381].log_data[1].valid := 1, [1381].log_data[2].valid := 1, [1381].log_data[3].valid := 1, [1381].log_data[4].valid := 1, [1381].log_data[5].valid := 1, [1381].log_data[6].valid := 1, [1381].log_data[7].valid := 1, [1381].log_data[8].valid := 1, [1381].log_data[9].valid := 1, [1381].log_data[10].valid := 1, [1381].log_data[11].valid := 1, [1381].log_data[12].valid := 1, [1381].log_data[13].valid := 1,
        [1381].log_data[14].valid := 1, [1381].log_data[15].valid := 1, [1381].log_data[16].valid := 1, [1381].log_data[17].valid := 1, [1381].log_data[18].valid := 1, [1381].log_data[19].valid := 1, [1381].time.Year := 2023, [1381].time.Month := 1, [1381].time.Day := 14, [1381].time.Hour := 11, [1381].time.Minute := 29, [1381].time.Second := 59, [1382].log_data[0].min := 1.0, [1382].log_data[0].max := 1.0, [1382].log_data[0].total := 300.0, [1382].log_data[0].time := 300.0, [1382].log_data[0].minminute := 30, [1382].log_data[0].maxminute := 30, [1382].log_data[0].valid := 1, [1382].log_data[1].valid := 1, [1382].log_data[2].valid := 1, [1382].log_data[3].valid := 1, [1382].log_data[4].valid := 1, [1382].log_data[5].valid := 1, [1382].log_data[6].valid := 1, [1382].log_data[7].valid := 1, [1382].log_data[8].valid := 1, [1382].log_data[9].valid := 1, [1382].log_data[10].valid := 1, [1382].log_data[11].valid := 1, [1382].log_data[12].valid := 1, [1382].log_data[13].valid := 1, [1382].log_data[14].valid := 1, [1382].log_data[15].valid := 1, [1382].log_data[16].valid := 1, [1382].log_data[17].valid := 1, [1382].log_data[18].valid := 1, [1382].log_data[19].valid := 1, [1382].time.Year := 2023, [1382].time.Month := 1, [1382].time.Day := 14, [1382].time.Hour := 11, [1382].time.Minute := 34, [1382].time.Second := 59, [1383].log_data[0].min := 1.0, [1383].log_data[0].max := 1.0, [1383].log_data[0].total := 300.0, [1383].log_data[0].time := 300.0, [1383].log_data[0].minminute := 35, [1383].log_data[0].maxminute := 35, [1383].log_data[0].valid := 1, [1383].log_data[1].valid := 1, [1383].log_data[2].valid := 1, [1383].log_data[3].valid := 1, [1383].log_data[4].valid := 1, [1383].log_data[5].valid := 1, [1383].log_data[6].valid := 1, [1383].log_data[7].valid := 1, [1383].log_data[8].valid := 1, [1383].log_data[9].valid := 1,
        [1383].log_data[10].valid := 1, [1383].log_data[11].valid := 1, [1383].log_data[12].valid := 1, [1383].log_data[13].valid := 1, [1383].log_data[14].valid := 1, [1383].log_data[15].valid := 1, [1383].log_data[16].valid := 1, [1383].log_data[17].valid := 1, [1383].log_data[18].valid := 1, [1383].log_data[19].valid := 1, [1383].time.Year := 2023, [1383].time.Month := 1, [1383].time.Day := 14, [1383].time.Hour := 11, [1383].time.Minute := 39, [1383].time.Second := 59, [1384].log_data[0].min := 1.0, [1384].log_data[0].max := 1.0, [1384].log_data[0].total := 300.0, [1384].log_data[0].time := 300.0, [1384].log_data[0].minminute := 40, [1384].log_data[0].maxminute := 40, [1384].log_data[0].valid := 1, [1384].log_data[1].valid := 1, [1384].log_data[2].valid := 1, [1384].log_data[3].valid := 1, [1384].log_data[4].valid := 1, [1384].log_data[5].valid := 1, [1384].log_data[6].valid := 1, [1384].log_data[7].valid := 1, [1384].log_data[8].valid := 1, [1384].log_data[9].valid := 1, [1384].log_data[10].valid := 1, [1384].log_data[11].valid := 1, [1384].log_data[12].valid := 1, [1384].log_data[13].valid := 1, [1384].log_data[14].valid := 1, [1384].log_data[15].valid := 1, [1384].log_data[16].valid := 1, [1384].log_data[17].valid := 1, [1384].log_data[18].valid := 1, [1384].log_data[19].valid := 1, [1384].time.Year := 2023, [1384].time.Month := 1, [1384].time.Day := 14, [1384].time.Hour := 11, [1384].time.Minute := 44, [1384].time.Second := 59, [1385].log_data[0].min := 1.0, [1385].log_data[0].max := 1.0, [1385].log_data[0].total := 300.0, [1385].log_data[0].time := 300.0, [1385].log_data[0].minminute := 45, [1385].log_data[0].maxminute := 45, [1385].log_data[0].valid := 1, [1385].log_data[1].valid := 1, [1385].log_data[2].valid := 1, [1385].log_data[3].valid := 1, [1385].log_data[4].valid := 1, [1385].log_data[5].valid := 1,
        [1385].log_data[6].valid := 1, [1385].log_data[7].valid := 1, [1385].log_data[8].valid := 1, [1385].log_data[9].valid := 1, [1385].log_data[10].valid := 1, [1385].log_data[11].valid := 1, [1385].log_data[12].valid := 1, [1385].log_data[13].valid := 1, [1385].log_data[14].valid := 1, [1385].log_data[15].valid := 1, [1385].log_data[16].valid := 1, [1385].log_data[17].valid := 1, [1385].log_data[18].valid := 1, [1385].log_data[19].valid := 1, [1385].time.Year := 2023, [1385].time.Month := 1, [1385].time.Day := 14, [1385].time.Hour := 11, [1385].time.Minute := 49, [1385].time.Second := 59, [1386].log_data[0].min := 1.0, [1386].log_data[0].max := 1.0, [1386].log_data[0].total := 300.0, [1386].log_data[0].time := 300.0, [1386].log_data[0].minminute := 50, [1386].log_data[0].maxminute := 50, [1386].log_data[0].valid := 1, [1386].log_data[1].valid := 1, [1386].log_data[2].valid := 1, [1386].log_data[3].valid := 1, [1386].log_data[4].valid := 1, [1386].log_data[5].valid := 1, [1386].log_data[6].valid := 1, [1386].log_data[7].valid := 1, [1386].log_data[8].valid := 1, [1386].log_data[9].valid := 1, [1386].log_data[10].valid := 1, [1386].log_data[11].valid := 1, [1386].log_data[12].valid := 1, [1386].log_data[13].valid := 1, [1386].log_data[14].valid := 1, [1386].log_data[15].valid := 1, [1386].log_data[16].valid := 1, [1386].log_data[17].valid := 1, [1386].log_data[18].valid := 1, [1386].log_data[19].valid := 1, [1386].time.Year := 2023, [1386].time.Month := 1, [1386].time.Day := 14, [1386].time.Hour := 11, [1386].time.Minute := 54, [1386].time.Second := 59, [1387].log_data[0].min := 1.0, [1387].log_data[0].max := 1.0, [1387].log_data[0].total := 300.0, [1387].log_data[0].time := 300.0, [1387].log_data[0].minminute := 55, [1387].log_data[0].maxminute := 55, [1387].log_data[0].valid := 1, [1387].log_data[1].valid := 1,
        [1387].log_data[2].valid := 1, [1387].log_data[3].valid := 1, [1387].log_data[4].valid := 1, [1387].log_data[5].valid := 1, [1387].log_data[6].valid := 1, [1387].log_data[7].valid := 1, [1387].log_data[8].valid := 1, [1387].log_data[9].valid := 1, [1387].log_data[10].valid := 1, [1387].log_data[11].valid := 1, [1387].log_data[12].valid := 1, [1387].log_data[13].valid := 1, [1387].log_data[14].valid := 1, [1387].log_data[15].valid := 1, [1387].log_data[16].valid := 1, [1387].log_data[17].valid := 1, [1387].log_data[18].valid := 1, [1387].log_data[19].valid := 1, [1387].time.Year := 2023, [1387].time.Month := 1, [1387].time.Day := 14, [1387].time.Hour := 11, [1387].time.Minute := 59, [1387].time.Second := 59, [1388].log_data[0].min := 1.0, [1388].log_data[0].max := 1.0, [1388].log_data[0].total := 299.5, [1388].log_data[0].time := 299.5, [1388].log_data[0].valid := 1, [1388].log_data[1].valid := 1, [1388].log_data[2].valid := 1, [1388].log_data[3].valid := 1, [1388].log_data[4].valid := 1, [1388].log_data[5].valid := 1, [1388].log_data[6].valid := 1, [1388].log_data[7].valid := 1, [1388].log_data[8].valid := 1, [1388].log_data[9].valid := 1, [1388].log_data[10].valid := 1, [1388].log_data[11].valid := 1, [1388].log_data[12].valid := 1, [1388].log_data[13].valid := 1, [1388].log_data[14].valid := 1, [1388].log_data[15].valid := 1, [1388].log_data[16].valid := 1, [1388].log_data[17].valid := 1, [1388].log_data[18].valid := 1, [1388].log_data[19].valid := 1, [1388].time.Year := 2023, [1388].time.Month := 1, [1388].time.Day := 14, [1388].time.Hour := 12, [1388].time.Minute := 4, [1388].time.Second := 59, [1389].log_data[0].min := 1.0, [1389].log_data[0].max := 1.0, [1389].log_data[0].total := 300.0, [1389].log_data[0].time := 300.0, [1389].log_data[0].minminute := 5, [1389].log_data[0].maxminute := 5,
        [1389].log_data[0].valid := 1, [1389].log_data[1].valid := 1, [1389].log_data[2].valid := 1, [1389].log_data[3].valid := 1, [1389].log_data[4].valid := 1, [1389].log_data[5].valid := 1, [1389].log_data[6].valid := 1, [1389].log_data[7].valid := 1, [1389].log_data[8].valid := 1, [1389].log_data[9].valid := 1, [1389].log_data[10].valid := 1, [1389].log_data[11].valid := 1, [1389].log_data[12].valid := 1, [1389].log_data[13].valid := 1, [1389].log_data[14].valid := 1, [1389].log_data[15].valid := 1, [1389].log_data[16].valid := 1, [1389].log_data[17].valid := 1, [1389].log_data[18].valid := 1, [1389].log_data[19].valid := 1, [1389].time.Year := 2023, [1389].time.Month := 1, [1389].time.Day := 14, [1389].time.Hour := 12, [1389].time.Minute := 9, [1389].time.Second := 59, [1390].log_data[0].min := 1.0, [1390].log_data[0].max := 1.0, [1390].log_data[0].total := 300.0, [1390].log_data[0].time := 300.0, [1390].log_data[0].minminute := 10, [1390].log_data[0].maxminute := 10, [1390].log_data[0].valid := 1, [1390].log_data[1].valid := 1, [1390].log_data[2].valid := 1, [1390].log_data[3].valid := 1, [1390].log_data[4].valid := 1, [1390].log_data[5].valid := 1, [1390].log_data[6].valid := 1, [1390].log_data[7].valid := 1, [1390].log_data[8].valid := 1, [1390].log_data[9].valid := 1, [1390].log_data[10].valid := 1, [1390].log_data[11].valid := 1, [1390].log_data[12].valid := 1, [1390].log_data[13].valid := 1, [1390].log_data[14].valid := 1, [1390].log_data[15].valid := 1, [1390].log_data[16].valid := 1, [1390].log_data[17].valid := 1, [1390].log_data[18].valid := 1, [1390].log_data[19].valid := 1, [1390].time.Year := 2023, [1390].time.Month := 1, [1390].time.Day := 14, [1390].time.Hour := 12, [1390].time.Minute := 14, [1390].time.Second := 59, [1391].log_data[0].min := 1.0, [1391].log_data[0].max := 1.0,
        [1391].log_data[0].total := 300.0, [1391].log_data[0].time := 300.0, [1391].log_data[0].minminute := 15, [1391].log_data[0].maxminute := 15, [1391].log_data[0].valid := 1, [1391].log_data[1].valid := 1, [1391].log_data[2].valid := 1, [1391].log_data[3].valid := 1, [1391].log_data[4].valid := 1, [1391].log_data[5].valid := 1, [1391].log_data[6].valid := 1, [1391].log_data[7].valid := 1, [1391].log_data[8].valid := 1, [1391].log_data[9].valid := 1, [1391].log_data[10].valid := 1, [1391].log_data[11].valid := 1, [1391].log_data[12].valid := 1, [1391].log_data[13].valid := 1, [1391].log_data[14].valid := 1, [1391].log_data[15].valid := 1, [1391].log_data[16].valid := 1, [1391].log_data[17].valid := 1, [1391].log_data[18].valid := 1, [1391].log_data[19].valid := 1, [1391].time.Year := 2023, [1391].time.Month := 1, [1391].time.Day := 14, [1391].time.Hour := 12, [1391].time.Minute := 19, [1391].time.Second := 59, [1392].log_data[0].min := 1.0, [1392].log_data[0].max := 1.0, [1392].log_data[0].total := 300.0, [1392].log_data[0].time := 300.0, [1392].log_data[0].minminute := 20, [1392].log_data[0].maxminute := 20, [1392].log_data[0].valid := 1, [1392].log_data[1].valid := 1, [1392].log_data[2].valid := 1, [1392].log_data[3].valid := 1, [1392].log_data[4].valid := 1, [1392].log_data[5].valid := 1, [1392].log_data[6].valid := 1, [1392].log_data[7].valid := 1, [1392].log_data[8].valid := 1, [1392].log_data[9].valid := 1, [1392].log_data[10].valid := 1, [1392].log_data[11].valid := 1, [1392].log_data[12].valid := 1, [1392].log_data[13].valid := 1, [1392].log_data[14].valid := 1, [1392].log_data[15].valid := 1, [1392].log_data[16].valid := 1, [1392].log_data[17].valid := 1, [1392].log_data[18].valid := 1, [1392].log_data[19].valid := 1, [1392].time.Year := 2023, [1392].time.Month := 1, [1392].time.Day := 14, [1392].time.Hour := 12,
        [1392].time.Minute := 24, [1392].time.Second := 59, [1393].log_data[0].min := 1.0, [1393].log_data[0].max := 1.0, [1393].log_data[0].total := 300.0, [1393].log_data[0].time := 300.0, [1393].log_data[0].minminute := 25, [1393].log_data[0].maxminute := 25, [1393].log_data[0].valid := 1, [1393].log_data[1].valid := 1, [1393].log_data[2].valid := 1, [1393].log_data[3].valid := 1, [1393].log_data[4].valid := 1, [1393].log_data[5].valid := 1, [1393].log_data[6].valid := 1, [1393].log_data[7].valid := 1, [1393].log_data[8].valid := 1, [1393].log_data[9].valid := 1, [1393].log_data[10].valid := 1, [1393].log_data[11].valid := 1, [1393].log_data[12].valid := 1, [1393].log_data[13].valid := 1, [1393].log_data[14].valid := 1, [1393].log_data[15].valid := 1, [1393].log_data[16].valid := 1, [1393].log_data[17].valid := 1, [1393].log_data[18].valid := 1, [1393].log_data[19].valid := 1, [1393].time.Year := 2023, [1393].time.Month := 1, [1393].time.Day := 14, [1393].time.Hour := 12, [1393].time.Minute := 29, [1393].time.Second := 59, [1394].log_data[0].min := 1.0, [1394].log_data[0].max := 1.0, [1394].log_data[0].total := 300.0, [1394].log_data[0].time := 300.0, [1394].log_data[0].minminute := 30, [1394].log_data[0].maxminute := 30, [1394].log_data[0].valid := 1, [1394].log_data[1].valid := 1, [1394].log_data[2].valid := 1, [1394].log_data[3].valid := 1, [1394].log_data[4].valid := 1, [1394].log_data[5].valid := 1, [1394].log_data[6].valid := 1, [1394].log_data[7].valid := 1, [1394].log_data[8].valid := 1, [1394].log_data[9].valid := 1, [1394].log_data[10].valid := 1, [1394].log_data[11].valid := 1, [1394].log_data[12].valid := 1, [1394].log_data[13].valid := 1, [1394].log_data[14].valid := 1, [1394].log_data[15].valid := 1, [1394].log_data[16].valid := 1, [1394].log_data[17].valid := 1, [1394].log_data[18].valid := 1, [1394].log_data[19].valid := 1,
        [1394].time.Year := 2023, [1394].time.Month := 1, [1394].time.Day := 14, [1394].time.Hour := 12, [1394].time.Minute := 34, [1394].time.Second := 59, [1395].log_data[0].min := 1.0, [1395].log_data[0].max := 1.0, [1395].log_data[0].total := 300.0, [1395].log_data[0].time := 300.0, [1395].log_data[0].minminute := 35, [1395].log_data[0].maxminute := 35, [1395].log_data[0].valid := 1, [1395].log_data[1].valid := 1, [1395].log_data[2].valid := 1, [1395].log_data[3].valid := 1, [1395].log_data[4].valid := 1, [1395].log_data[5].valid := 1, [1395].log_data[6].valid := 1, [1395].log_data[7].valid := 1, [1395].log_data[8].valid := 1, [1395].log_data[9].valid := 1, [1395].log_data[10].valid := 1, [1395].log_data[11].valid := 1, [1395].log_data[12].valid := 1, [1395].log_data[13].valid := 1, [1395].log_data[14].valid := 1, [1395].log_data[15].valid := 1, [1395].log_data[16].valid := 1, [1395].log_data[17].valid := 1, [1395].log_data[18].valid := 1, [1395].log_data[19].valid := 1, [1395].time.Year := 2023, [1395].time.Month := 1, [1395].time.Day := 14, [1395].time.Hour := 12, [1395].time.Minute := 39, [1395].time.Second := 59, [1396].log_data[0].min := 1.0, [1396].log_data[0].max := 1.0, [1396].log_data[0].total := 300.0, [1396].log_data[0].time := 300.0, [1396].log_data[0].minminute := 40, [1396].log_data[0].maxminute := 40, [1396].log_data[0].valid := 1, [1396].log_data[1].valid := 1, [1396].log_data[2].valid := 1, [1396].log_data[3].valid := 1, [1396].log_data[4].valid := 1, [1396].log_data[5].valid := 1, [1396].log_data[6].valid := 1, [1396].log_data[7].valid := 1, [1396].log_data[8].valid := 1, [1396].log_data[9].valid := 1, [1396].log_data[10].valid := 1, [1396].log_data[11].valid := 1, [1396].log_data[12].valid := 1, [1396].log_data[13].valid := 1, [1396].log_data[14].valid := 1, [1396].log_data[15].valid := 1,
        [1396].log_data[16].valid := 1, [1396].log_data[17].valid := 1, [1396].log_data[18].valid := 1, [1396].log_data[19].valid := 1, [1396].time.Year := 2023, [1396].time.Month := 1, [1396].time.Day := 14, [1396].time.Hour := 12, [1396].time.Minute := 44, [1396].time.Second := 59, [1397].log_data[0].min := 1.0, [1397].log_data[0].max := 1.0, [1397].log_data[0].total := 300.0, [1397].log_data[0].time := 300.0, [1397].log_data[0].minminute := 45, [1397].log_data[0].maxminute := 45, [1397].log_data[0].valid := 1, [1397].log_data[1].valid := 1, [1397].log_data[2].valid := 1, [1397].log_data[3].valid := 1, [1397].log_data[4].valid := 1, [1397].log_data[5].valid := 1, [1397].log_data[6].valid := 1, [1397].log_data[7].valid := 1, [1397].log_data[8].valid := 1, [1397].log_data[9].valid := 1, [1397].log_data[10].valid := 1, [1397].log_data[11].valid := 1, [1397].log_data[12].valid := 1, [1397].log_data[13].valid := 1, [1397].log_data[14].valid := 1, [1397].log_data[15].valid := 1, [1397].log_data[16].valid := 1, [1397].log_data[17].valid := 1, [1397].log_data[18].valid := 1, [1397].log_data[19].valid := 1, [1397].time.Year := 2023, [1397].time.Month := 1, [1397].time.Day := 14, [1397].time.Hour := 12, [1397].time.Minute := 49, [1397].time.Second := 59, [1398].log_data[0].min := 1.0, [1398].log_data[0].max := 1.0, [1398].log_data[0].total := 300.0, [1398].log_data[0].time := 300.0, [1398].log_data[0].minminute := 50, [1398].log_data[0].maxminute := 50, [1398].log_data[0].valid := 1, [1398].log_data[1].valid := 1, [1398].log_data[2].valid := 1, [1398].log_data[3].valid := 1, [1398].log_data[4].valid := 1, [1398].log_data[5].valid := 1, [1398].log_data[6].valid := 1, [1398].log_data[7].valid := 1, [1398].log_data[8].valid := 1, [1398].log_data[9].valid := 1, [1398].log_data[10].valid := 1, [1398].log_data[11].valid := 1,
        [1398].log_data[12].valid := 1, [1398].log_data[13].valid := 1, [1398].log_data[14].valid := 1, [1398].log_data[15].valid := 1, [1398].log_data[16].valid := 1, [1398].log_data[17].valid := 1, [1398].log_data[18].valid := 1, [1398].log_data[19].valid := 1, [1398].time.Year := 2023, [1398].time.Month := 1, [1398].time.Day := 14, [1398].time.Hour := 12, [1398].time.Minute := 54, [1398].time.Second := 59, [1399].log_data[0].min := 1.0, [1399].log_data[0].max := 1.0, [1399].log_data[0].total := 300.0, [1399].log_data[0].time := 300.0, [1399].log_data[0].minminute := 55, [1399].log_data[0].maxminute := 55, [1399].log_data[0].valid := 1, [1399].log_data[1].valid := 1, [1399].log_data[2].valid := 1, [1399].log_data[3].valid := 1, [1399].log_data[4].valid := 1, [1399].log_data[5].valid := 1, [1399].log_data[6].valid := 1, [1399].log_data[7].valid := 1, [1399].log_data[8].valid := 1, [1399].log_data[9].valid := 1, [1399].log_data[10].valid := 1, [1399].log_data[11].valid := 1, [1399].log_data[12].valid := 1, [1399].log_data[13].valid := 1, [1399].log_data[14].valid := 1, [1399].log_data[15].valid := 1, [1399].log_data[16].valid := 1, [1399].log_data[17].valid := 1, [1399].log_data[18].valid := 1, [1399].log_data[19].valid := 1, [1399].time.Year := 2023, [1399].time.Month := 1, [1399].time.Day := 14, [1399].time.Hour := 12, [1399].time.Minute := 59, [1399].time.Second := 59, [1400].log_data[0].min := 1.0, [1400].log_data[0].max := 1.0, [1400].log_data[0].total := 300.0, [1400].log_data[0].time := 300.0, [1400].log_data[0].valid := 1, [1400].log_data[1].valid := 1, [1400].log_data[2].valid := 1, [1400].log_data[3].valid := 1, [1400].log_data[4].valid := 1, [1400].log_data[5].valid := 1, [1400].log_data[6].valid := 1, [1400].log_data[7].valid := 1, [1400].log_data[8].valid := 1, [1400].log_data[9].valid := 1,
        [1400].log_data[10].valid := 1, [1400].log_data[11].valid := 1, [1400].log_data[12].valid := 1, [1400].log_data[13].valid := 1, [1400].log_data[14].valid := 1, [1400].log_data[15].valid := 1, [1400].log_data[16].valid := 1, [1400].log_data[17].valid := 1, [1400].log_data[18].valid := 1, [1400].log_data[19].valid := 1, [1400].time.Year := 2023, [1400].time.Month := 1, [1400].time.Day := 14, [1400].time.Hour := 13, [1400].time.Minute := 4, [1400].time.Second := 59, [1401].log_data[0].min := 1.0, [1401].log_data[0].max := 1.0, [1401].log_data[0].total := 300.0, [1401].log_data[0].time := 300.0, [1401].log_data[0].minminute := 5, [1401].log_data[0].maxminute := 5, [1401].log_data[0].valid := 1, [1401].log_data[1].valid := 1, [1401].log_data[2].valid := 1, [1401].log_data[3].valid := 1, [1401].log_data[4].valid := 1, [1401].log_data[5].valid := 1, [1401].log_data[6].valid := 1, [1401].log_data[7].valid := 1, [1401].log_data[8].valid := 1, [1401].log_data[9].valid := 1, [1401].log_data[10].valid := 1, [1401].log_data[11].valid := 1, [1401].log_data[12].valid := 1, [1401].log_data[13].valid := 1, [1401].log_data[14].valid := 1, [1401].log_data[15].valid := 1, [1401].log_data[16].valid := 1, [1401].log_data[17].valid := 1, [1401].log_data[18].valid := 1, [1401].log_data[19].valid := 1, [1401].time.Year := 2023, [1401].time.Month := 1, [1401].time.Day := 14, [1401].time.Hour := 13, [1401].time.Minute := 9, [1401].time.Second := 59, [1402].log_data[0].min := 1.0, [1402].log_data[0].max := 1.0, [1402].log_data[0].total := 300.0, [1402].log_data[0].time := 300.0, [1402].log_data[0].minminute := 10, [1402].log_data[0].maxminute := 10, [1402].log_data[0].valid := 1, [1402].log_data[1].valid := 1, [1402].log_data[2].valid := 1, [1402].log_data[3].valid := 1, [1402].log_data[4].valid := 1, [1402].log_data[5].valid := 1,
